	X =  248.562  mm,	Y =   -335.401  mm,	Z =   -309.100  mm,
	W =  90.000 deg,	P =   0.000 deg,	R =   90.000 deg
};
P[1872]{
   GP1:
	UF : 0, UT : 6,		CONFIG : 'N U T, 0, 0, 0',
	X =  247.422  mm,	Y =   -335.745  mm,	Z =   -309.000  mm,
	W =  90.000 deg,	P =   0.000 deg,	R =   90.000 deg
};
P[1873]{
   GP1:
	UF : 0, UT : 6,		CONFIG : 'N U T, 0, 0, 0',
	X =  247.235  mm,	Y =   -336.680  mm,	Z =   -320.106  mm,
	W =  90.000 deg,	P =   0.000 deg,	R =   90.000 deg
};
P[1874]{
   GP1:
	UF : 0, UT : 6,		CONFIG : 'N U T, 0, 0, 0',
	X =  245.967  mm,	Y =   -336.637  mm,	Z =   -309.000  mm,
	W =  90.000 deg,	P =   0.000 deg,	R =   90.000 deg
};
P[1875]{
   GP1:
	UF : 0, UT : 6,		CONFIG : 'N U T, 0, 0, 0',
	X =  245.051  mm,	Y =   -337.530  mm,	Z =   -309.000  mm,
	W =  90.000 deg,	P =   0.000 deg,	R =   90.000 deg
};
P[1876]{
   GP1:
	UF : 0, UT : 6,		CONFIG : 'N U T, 0, 0, 0',
	X =  243.808  mm,	Y =   -338.459  mm,	Z =   -309.000  mm,
	W =  90.000 deg,	P =   0.000 deg,	R =   90.000 deg
};
P[1877]{
   GP1:
	UF : 0, UT : 6,		CONFIG : 'N U T, 0, 0, 0',
	X =  242.999  mm,	Y =   -338.641  mm,	Z =   -309.100  mm,
	W =  90.000 deg,	P =   0.000 deg,	R =   90.000 deg
};
P[1878]{
   GP1:
	UF : 0, UT : 6,		CONFIG : 'N U T, 0, 0, 0',
	X =  242.520  mm,	Y =   -339.408  mm,	Z =   -309.100  mm,
	W =  90.000 deg,	P =   0.000 deg,	R =   90.000 deg
};
P[1879]{
   GP1:
	UF : 0, UT : 6,		CONFIG : 'N U T, 0, 0, 0',
	X =  240.721  mm,	Y =   -340.006  mm,	Z =   -309.100  mm,
	W =  90.000 deg,	P =   0.000 deg,	R =   90.000 deg
};
P[1880]{
   GP1:
	UF : 0, UT : 6,		CONFIG : 'N U T, 0, 0, 0',
	X =  239.710  mm,	Y =   -340.345  mm,	Z =   -309.000  mm,
	W =  90.000 deg,	P =   0.000 deg,	R =   90.000 deg
};
P[1881]{
   GP1:
	UF : 0, UT : 6,		CONFIG : 'N U T, 0, 0, 0',
	X =  238.388  mm,	Y =   -341.396  mm,	Z =   -309.000  mm,
	W =  90.000 deg,	P =   0.000 deg,	R =   90.000 deg
};
P[1882]{
   GP1:
	UF : 0, UT : 6,		CONFIG : 'N U T, 0, 0, 0',
	X =  236.976  mm,	Y =   -342.451  mm,	Z =   -309.000  mm,
	W =  90.000 deg,	P =   0.000 deg,	R =   90.000 deg
};
P[1883]{
   GP1:
	UF : 0, UT : 6,		CONFIG : 'N U T, 0, 0, 0',
	X =  236.149  mm,	Y =   -342.418  mm,	Z =   -309.100  mm,
	W =  90.000 deg,	P =   0.000 deg,	R =   90.000 deg
};
P[1884]{
   GP1:
	UF : 0, UT : 6,		CONFIG : 'N U T, 0, 0, 0',
	X =  235.257  mm,	Y =   -343.142  mm,	Z =   -328.083  mm,
	W =  90.000 deg,	P =   0.000 deg,	R =   90.000 deg
};
P[1885]{
   GP1:
	UF : 0, UT : 6,		CONFIG : 'N U T, 0, 0, 0',
	X =  233.924  mm,	Y =   -343.541  mm,	Z =   -309.100  mm,
	W =  90.000 deg,	P =   0.000 deg,	R =   90.000 deg
};
P[1886]{
   GP1:
	UF : 0, UT : 6,		CONFIG : 'N U T, 0, 0, 0',
	X =  232.946  mm,	Y =   -344.617  mm,	Z =   -309.000  mm,
	W =  90.000 deg,	P =   0.000 deg,	R =   90.000 deg
};
P[1887]{
   GP1:
	UF : 0, UT : 6,		CONFIG : 'N U T, 0, 0, 0',
	X =  231.730  mm,	Y =   -344.591  mm,	Z =   -309.000  mm,
	W =  90.000 deg,	P =   0.000 deg,	R =   90.000 deg
};
P[1888]{
   GP1:
	UF : 0, UT : 6,		CONFIG : 'N U T, 0, 0, 0',
	X =  231.106  mm,	Y =   -345.617  mm,	Z =   -309.100  mm,
	W =  90.000 deg,	P =   0.000 deg,	R =   90.000 deg
};
P[1889]{
   GP1:
	UF : 0, UT : 6,		CONFIG : 'N U T, 0, 0, 0',
	X =  229.581  mm,	Y =   -346.237  mm,	Z =   -309.000  mm,
	W =  90.000 deg,	P =   0.000 deg,	R =   90.000 deg
};
P[1890]{
   GP1:
	UF : 0, UT : 6,		CONFIG : 'N U T, 0, 0, 0',
	X =  228.460  mm,	Y =   -346.775  mm,	Z =   -309.000  mm,
	W =  90.000 deg,	P =   0.000 deg,	R =   90.000 deg
};
P[1891]{
   GP1:
	UF : 0, UT : 6,		CONFIG : 'N U T, 0, 0, 0',
	X =  227.482  mm,	Y =   -347.579  mm,	Z =   -309.000  mm,
	W =  90.000 deg,	P =   0.000 deg,	R =   90.000 deg
};
P[1892]{
   GP1:
	UF : 0, UT : 6,		CONFIG : 'N U T, 0, 0, 0',
	X =  226.728  mm,	Y =   -348.283  mm,	Z =   -309.000  mm,
	W =  90.000 deg,	P =   0.000 deg,	R =   90.000 deg
};
P[1893]{
   GP1:
	UF : 0, UT : 6,		CONFIG : 'N U T, 0, 0, 0',
	X =  225.408  mm,	Y =   -348.579  mm,	Z =   -309.000  mm,
	W =  90.000 deg,	P =   0.000 deg,	R =   90.000 deg
};
P[1894]{
   GP1:
	UF : 0, UT : 6,		CONFIG : 'N U T, 0, 0, 0',
	X =  224.991  mm,	Y =   -349.488  mm,	Z =   -309.100  mm,
	W =  90.000 deg,	P =   0.000 deg,	R =   90.000 deg
};
P[1895]{
   GP1:
	UF : 0, UT : 6,		CONFIG : 'N U T, 0, 0, 0',
	X =  223.968  mm,	Y =   -349.539  mm,	Z =   -309.000  mm,
	W =  90.000 deg,	P =   0.000 deg,	R =   90.000 deg
};
P[1896]{
   GP1:
	UF : 0, UT : 6,		CONFIG : 'N U T, 0, 0, 0',
	X =  223.129  mm,	Y =   -350.051  mm,	Z =   -314.213  mm,
	W =  90.000 deg,	P =   0.000 deg,	R =   90.000 deg
};
P[1897]{
   GP1:
	UF : 0, UT : 6,		CONFIG : 'N U T, 0, 0, 0',
	X =  222.469  mm,	Y =   -350.654  mm,	Z =   -309.577  mm,
	W =  90.000 deg,	P =   0.000 deg,	R =   90.000 deg
};
P[1898]{
   GP1:
	UF : 0, UT : 6,		CONFIG : 'N U T, 0, 0, 0',
	X =  221.386  mm,	Y =   -350.938  mm,	Z =   -309.100  mm,
	W =  90.000 deg,	P =   0.000 deg,	R =   90.000 deg
};
P[1899]{
   GP1:
	UF : 0, UT : 6,		CONFIG : 'N U T, 0, 0, 0',
	X =  220.623  mm,	Y =   -351.619  mm,	Z =   -309.000  mm,
	W =  90.000 deg,	P =   0.000 deg,	R =   90.000 deg
};
P[1900]{
   GP1:
	UF : 0, UT : 6,		CONFIG : 'N U T, 0, 0, 0',
	X =  219.642  mm,	Y =   -352.592  mm,	Z =   -321.382  mm,
	W =  90.000 deg,	P =   0.000 deg,	R =   90.000 deg
};
P[1901]{
   GP1:
	UF : 0, UT : 6,		CONFIG : 'N U T, 0, 0, 0',
	X =  218.872  mm,	Y =   -352.238  mm,	Z =   -309.000  mm,
	W =  90.000 deg,	P =   0.000 deg,	R =   90.000 deg
};
P[1902]{
   GP1:
	UF : 0, UT : 6,		CONFIG : 'N U T, 0, 0, 0',
	X =  218.325  mm,	Y =   -353.159  mm,	Z =   -309.000  mm,
	W =  90.000 deg,	P =   0.000 deg,	R =   90.000 deg
};
P[1903]{
   GP1:
	UF : 0, UT : 6,		CONFIG : 'N U T, 0, 0, 0',
	X =  217.117  mm,	Y =   -353.353  mm,	Z =   -309.000  mm,
	W =  90.000 deg,	P =   0.000 deg,	R =   90.000 deg
};
P[1904]{
   GP1:
	UF : 0, UT : 6,		CONFIG : 'N U T, 0, 0, 0',
	X =  216.830  mm,	Y =   -354.032  mm,	Z =   -309.000  mm,
	W =  90.000 deg,	P =   0.000 deg,	R =   90.000 deg
};
P[1905]{
   GP1:
	UF : 0, UT : 6,		CONFIG : 'N U T, 0, 0, 0',
	X =  215.180  mm,	Y =   -354.468  mm,	Z =   -317.962  mm,
	W =  90.000 deg,	P =   0.000 deg,	R =   90.000 deg
};
P[1906]{
   GP1:
	UF : 0, UT : 6,		CONFIG : 'N U T, 0, 0, 0',
	X =  213.998  mm,	Y =   -355.496  mm,	Z =   -309.000  mm,
	W =  90.000 deg,	P =   0.000 deg,	R =   90.000 deg
};
P[1907]{
   GP1:
	UF : 0, UT : 6,		CONFIG : 'N U T, 0, 0, 0',
	X =  212.895  mm,	Y =   -355.957  mm,	Z =   -309.000  mm,
	W =  90.000 deg,	P =   0.000 deg,	R =   90.000 deg
};
P[1908]{
   GP1:
	UF : 0, UT : 6,		CONFIG : 'N U T, 0, 0, 0',
	X =  212.166  mm,	Y =   -356.433  mm,	Z =   -309.100  mm,
	W =  90.000 deg,	P =   0.000 deg,	R =   90.000 deg
};
P[1909]{
   GP1:
	UF : 0, UT : 6,		CONFIG : 'N U T, 0, 0, 0',
	X =  211.060  mm,	Y =   -356.896  mm,	Z =   -309.100  mm,
	W =  90.000 deg,	P =   0.000 deg,	R =   90.000 deg
};
P[1910]{
   GP1:
	UF : 0, UT : 6,		CONFIG : 'N U T, 0, 0, 0',
	X =  209.472  mm,	Y =   -358.263  mm,	Z =   -309.000  mm,
	W =  90.000 deg,	P =   0.000 deg,	R =   90.000 deg
};
P[1911]{
   GP1:
	UF : 0, UT : 6,		CONFIG : 'N U T, 0, 0, 0',
	X =  208.197  mm,	Y =   -358.550  mm,	Z =   -309.000  mm,
	W =  90.000 deg,	P =   0.000 deg,	R =   90.000 deg
};
P[1912]{
   GP1:
	UF : 0, UT : 6,		CONFIG : 'N U T, 0, 0, 0',
	X =  207.007  mm,	Y =   -359.434  mm,	Z =   -309.000  mm,
	W =  90.000 deg,	P =   0.000 deg,	R =   90.000 deg
};
P[1913]{
   GP1:
	UF : 0, UT : 6,		CONFIG : 'N U T, 0, 0, 0',
	X =  206.131  mm,	Y =   -360.046  mm,	Z =   -309.000  mm,
	W =  90.000 deg,	P =   0.000 deg,	R =   90.000 deg
};
P[1914]{
   GP1:
	UF : 0, UT : 6,		CONFIG : 'N U T, 0, 0, 0',
	X =  205.000  mm,	Y =   -360.301  mm,	Z =   -309.100  mm,
	W =  90.000 deg,	P =   0.000 deg,	R =   90.000 deg
};
P[1915]{
   GP1:
	UF : 0, UT : 6,		CONFIG : 'N U T, 0, 0, 0',
	X =  204.421  mm,	Y =   -361.260  mm,	Z =   -309.000  mm,
	W =  90.000 deg,	P =   0.000 deg,	R =   90.000 deg
};
P[1916]{
   GP1:
	UF : 0, UT : 6,		CONFIG : 'N U T, 0, 0, 0',
	X =  202.482  mm,	Y =   -361.984  mm,	Z =   -309.100  mm,
	W =  90.000 deg,	P =   0.000 deg,	R =   90.000 deg
};
P[1917]{
   GP1:
	UF : 0, UT : 6,		CONFIG : 'N U T, 0, 0, 0',
	X =  201.337  mm,	Y =   -362.133  mm,	Z =   -309.115  mm,
	W =  90.000 deg,	P =   0.000 deg,	R =   90.000 deg
};
P[1918]{
   GP1:
	UF : 0, UT : 6,		CONFIG : 'N U T, 0, 0, 0',
	X =  200.951  mm,	Y =   -362.839  mm,	Z =   -309.100  mm,
	W =  90.000 deg,	P =   0.000 deg,	R =   90.000 deg
};
P[1919]{
   GP1:
	UF : 0, UT : 6,		CONFIG : 'N U T, 0, 0, 0',
	X =  199.770  mm,	Y =   -363.436  mm,	Z =   -309.100  mm,
	W =  90.000 deg,	P =   0.000 deg,	R =   90.000 deg
};
P[1920]{
   GP1:
	UF : 0, UT : 6,		CONFIG : 'N U T, 0, 0, 0',
	X =  198.938  mm,	Y =   -363.987  mm,	Z =   -309.100  mm,
	W =  90.000 deg,	P =   0.000 deg,	R =   90.000 deg
};
P[1921]{
   GP1:
	UF : 0, UT : 6,		CONFIG : 'N U T, 0, 0, 0',
	X =  198.274  mm,	Y =   -364.327  mm,	Z =   -309.000  mm,
	W =  90.000 deg,	P =   0.000 deg,	R =   90.000 deg
};
P[1922]{
   GP1:
	UF : 0, UT : 6,		CONFIG : 'N U T, 0, 0, 0',
	X =  197.346  mm,	Y =   -364.943  mm,	Z =   -313.498  mm,
	W =  90.000 deg,	P =   0.000 deg,	R =   90.000 deg
};
P[1923]{
   GP1:
	UF : 0, UT : 6,		CONFIG : 'N U T, 0, 0, 0',
	X =  196.755  mm,	Y =   -365.858  mm,	Z =   -309.000  mm,
	W =  90.000 deg,	P =   0.000 deg,	R =   90.000 deg
};
P[1924]{
   GP1:
	UF : 0, UT : 6,		CONFIG : 'N U T, 0, 0, 0',
	X =  196.093  mm,	Y =   -366.179  mm,	Z =   -309.000  mm,
	W =  90.000 deg,	P =   0.000 deg,	R =   90.000 deg
};
P[1925]{
   GP1:
	UF : 0, UT : 6,		CONFIG : 'N U T, 0, 0, 0',
	X =  194.785  mm,	Y =   -366.104  mm,	Z =   -309.100  mm,
	W =  90.000 deg,	P =   0.000 deg,	R =   90.000 deg
};
P[1926]{
   GP1:
	UF : 0, UT : 6,		CONFIG : 'N U T, 0, 0, 0',
	X =  193.345  mm,	Y =   -367.474  mm,	Z =   -309.000  mm,
	W =  90.000 deg,	P =   0.000 deg,	R =   90.000 deg
};
P[1927]{
   GP1:
	UF : 0, UT : 6,		CONFIG : 'N U T, 0, 0, 0',
	X =  192.179  mm,	Y =   -367.513  mm,	Z =   -316.834  mm,
	W =  90.000 deg,	P =   0.000 deg,	R =   90.000 deg
};
P[1928]{
   GP1:
	UF : 0, UT : 6,		CONFIG : 'N U T, 0, 0, 0',
	X =  191.363  mm,	Y =   -368.920  mm,	Z =   -318.857  mm,
	W =  90.000 deg,	P =   0.000 deg,	R =   90.000 deg
};
P[1929]{
   GP1:
	UF : 0, UT : 6,		CONFIG : 'N U T, 0, 0, 0',
	X =  190.046  mm,	Y =   -369.124  mm,	Z =   -309.000  mm,
	W =  90.000 deg,	P =   0.000 deg,	R =   90.000 deg
};
P[1930]{
   GP1:
	UF : 0, UT : 6,		CONFIG : 'N U T, 0, 0, 0',
	X =  188.428  mm,	Y =   -369.682  mm,	Z =   -309.000  mm,
	W =  90.000 deg,	P =   0.000 deg,	R =   90.000 deg
};
P[1931]{
   GP1:
	UF : 0, UT : 6,		CONFIG : 'N U T, 0, 0, 0',
	X =  187.625  mm,	Y =   -370.456  mm,	Z =   -309.000  mm,
	W =  90.000 deg,	P =   0.000 deg,	R =   90.000 deg
};
P[1932]{
   GP1:
	UF : 0, UT : 6,		CONFIG : 'N U T, 0, 0, 0',
	X =  186.427  mm,	Y =   -371.699  mm,	Z =   -312.203  mm,
	W =  90.000 deg,	P =   0.000 deg,	R =   90.000 deg
};
P[1933]{
   GP1:
	UF : 0, UT : 6,		CONFIG : 'N U T, 0, 0, 0',
	X =  185.466  mm,	Y =   -371.863  mm,	Z =   -309.100  mm,
	W =  90.000 deg,	P =   0.000 deg,	R =   90.000 deg
};
P[1934]{
   GP1:
	UF : 0, UT : 6,		CONFIG : 'N U T, 0, 0, 0',
	X =  184.245  mm,	Y =   -372.318  mm,	Z =   -309.000  mm,
	W =  90.000 deg,	P =   0.000 deg,	R =   90.000 deg
};
P[1935]{
   GP1:
	UF : 0, UT : 6,		CONFIG : 'N U T, 0, 0, 0',
	X =  183.685  mm,	Y =   -372.780  mm,	Z =   -309.100  mm,
	W =  90.000 deg,	P =   0.000 deg,	R =   90.000 deg
};
P[1936]{
   GP1:
	UF : 0, UT : 6,		CONFIG : 'N U T, 0, 0, 0',
	X =  183.047  mm,	Y =   -373.648  mm,	Z =   -309.000  mm,
	W =  90.000 deg,	P =   0.000 deg,	R =   90.000 deg
};
P[1937]{
   GP1:
	UF : 0, UT : 6,		CONFIG : 'N U T, 0, 0, 0',
	X =  182.264  mm,	Y =   -374.207  mm,	Z =   -309.000  mm,
	W =  90.000 deg,	P =   0.000 deg,	R =   90.000 deg
};
P[1938]{
   GP1:
	UF : 0, UT : 6,		CONFIG : 'N U T, 0, 0, 0',
	X =  180.861  mm,	Y =   -374.555  mm,	Z =   -309.000  mm,
	W =  90.000 deg,	P =   0.000 deg,	R =   90.000 deg
};
P[1939]{
   GP1:
	UF : 0, UT : 6,		CONFIG : 'N U T, 0, 0, 0',
	X =  180.053  mm,	Y =   -374.605  mm,	Z =   -309.000  mm,
	W =  90.000 deg,	P =   0.000 deg,	R =   90.000 deg
};
P[1940]{
   GP1:
	UF : 0, UT : 6,		CONFIG : 'N U T, 0, 0, 0',
	X =  178.977  mm,	Y =   -375.401  mm,	Z =   -309.000  mm,
	W =  90.000 deg,	P =   0.000 deg,	R =   90.000 deg
};
P[1941]{
   GP1:
	UF : 0, UT : 6,		CONFIG : 'N U T, 0, 0, 0',
	X =  178.071  mm,	Y =   -375.997  mm,	Z =   -309.100  mm,
	W =  90.000 deg,	P =   0.000 deg,	R =   90.000 deg
};
P[1942]{
   GP1:
	UF : 0, UT : 6,		CONFIG : 'N U T, 0, 0, 0',
	X =  176.472  mm,	Y =   -376.780  mm,	Z =   -319.410  mm,
	W =  90.000 deg,	P =   0.000 deg,	R =   90.000 deg
};
P[1943]{
   GP1:
	UF : 0, UT : 6,		CONFIG : 'N U T, 0, 0, 0',
	X =  175.518  mm,	Y =   -377.434  mm,	Z =   -318.225  mm,
	W =  90.000 deg,	P =   0.000 deg,	R =   90.000 deg
};
P[1944]{
   GP1:
	UF : 0, UT : 6,		CONFIG : 'N U T, 0, 0, 0',
	X =  174.768  mm,	Y =   -377.867  mm,	Z =   -309.100  mm,
	W =  90.000 deg,	P =   0.000 deg,	R =   90.000 deg
};
P[1945]{
   GP1:
	UF : 0, UT : 6,		CONFIG : 'N U T, 0, 0, 0',
	X =  174.000  mm,	Y =   -377.913  mm,	Z =   -309.000  mm,
	W =  90.000 deg,	P =   0.000 deg,	R =   90.000 deg
};
P[1946]{
   GP1:
	UF : 0, UT : 6,		CONFIG : 'N U T, 0, 0, 0',
	X =  173.393  mm,	Y =   -378.705  mm,	Z =   -309.100  mm,
	W =  90.000 deg,	P =   0.000 deg,	R =   90.000 deg
};
P[1947]{
   GP1:
	UF : 0, UT : 6,		CONFIG : 'N U T, 0, 0, 0',
	X =  172.740  mm,	Y =   -379.505  mm,	Z =   -309.000  mm,
	W =  90.000 deg,	P =   0.000 deg,	R =   90.000 deg
};
P[1948]{
   GP1:
	UF : 0, UT : 6,		CONFIG : 'N U T, 0, 0, 0',
	X =  171.553  mm,	Y =   -379.511  mm,	Z =   -309.000  mm,
	W =  90.000 deg,	P =   0.000 deg,	R =   90.000 deg
};
P[1949]{
   GP1:
	UF : 0, UT : 6,		CONFIG : 'N U T, 0, 0, 0',
	X =  170.266  mm,	Y =   -380.690  mm,	Z =   -309.100  mm,
	W =  90.000 deg,	P =   0.000 deg,	R =   90.000 deg
};
P[1950]{
   GP1:
	UF : 0, UT : 6,		CONFIG : 'N U T, 0, 0, 0',
	X =  169.463  mm,	Y =   -381.050  mm,	Z =   -309.100  mm,
	W =  90.000 deg,	P =   0.000 deg,	R =   90.000 deg
};
P[1951]{
   GP1:
	UF : 0, UT : 6,		CONFIG : 'N U T, 0, 0, 0',
	X =  168.875  mm,	Y =   -381.396  mm,	Z =   -309.000  mm,
	W =  90.000 deg,	P =   0.000 deg,	R =   90.000 deg
};
P[1952]{
   GP1:
	UF : 0, UT : 6,		CONFIG : 'N U T, 0, 0, 0',
	X =  168.134  mm,	Y =   -381.604  mm,	Z =   -309.100  mm,
	W =  90.000 deg,	P =   0.000 deg,	R =   90.000 deg
};
P[1953]{
   GP1:
	UF : 0, UT : 6,		CONFIG : 'N U T, 0, 0, 0',
	X =  167.049  mm,	Y =   -382.254  mm,	Z =   -309.000  mm,
	W =  90.000 deg,	P =   0.000 deg,	R =   90.000 deg
};
P[1954]{
   GP1:
	UF : 0, UT : 6,		CONFIG : 'N U T, 0, 0, 0',
	X =  166.356  mm,	Y =   -382.864  mm,	Z =   -319.959  mm,
	W =  90.000 deg,	P =   0.000 deg,	R =   90.000 deg
};
P[1955]{
   GP1:
	UF : 0, UT : 6,		CONFIG : 'N U T, 0, 0, 0',
	X =  165.358  mm,	Y =   -383.111  mm,	Z =   -309.100  mm,
	W =  90.000 deg,	P =   0.000 deg,	R =   90.000 deg
};
P[1956]{
   GP1:
	UF : 0, UT : 6,		CONFIG : 'N U T, 0, 0, 0',
	X =  164.331  mm,	Y =   -384.035  mm,	Z =   -309.000  mm,
	W =  90.000 deg,	P =   0.000 deg,	R =   90.000 deg
};
P[1957]{
   GP1:
	UF : 0, UT : 6,		CONFIG : 'N U T, 0, 0, 0',
	X =  163.613  mm,	Y =   -384.424  mm,	Z =   -309.100  mm,
	W =  90.000 deg,	P =   0.000 deg,	R =   90.000 deg
};
P[1958]{
   GP1:
	UF : 0, UT : 6,		CONFIG : 'N U T, 0, 0, 0',
	X =  162.736  mm,	Y =   -384.918  mm,	Z =   -309.100  mm,
	W =  90.000 deg,	P =   0.000 deg,	R =   90.000 deg
};
P[1959]{
   GP1:
	UF : 0, UT : 6,		CONFIG : 'N U T, 0, 0, 0',
	X =  162.209  mm,	Y =   -385.446  mm,	Z =   -309.050  mm,
	W =  90.000 deg,	P =   0.000 deg,	R =   90.000 deg
};
P[1960]{
   GP1:
	UF : 0, UT : 6,		CONFIG : 'N U T, 0, 0, 0',
	X =  160.970  mm,	Y =   -386.136  mm,	Z =   -309.000  mm,
	W =  90.000 deg,	P =   0.000 deg,	R =   90.000 deg
};
P[1961]{
   GP1:
	UF : 0, UT : 6,		CONFIG : 'N U T, 0, 0, 0',
	X =  159.328  mm,	Y =   -386.935  mm,	Z =   -317.393  mm,
	W =  90.000 deg,	P =   0.000 deg,	R =   90.000 deg
};
P[1962]{
   GP1:
	UF : 0, UT : 6,		CONFIG : 'N U T, 0, 0, 0',
	X =  158.454  mm,	Y =   -387.478  mm,	Z =   -309.000  mm,
	W =  90.000 deg,	P =   0.000 deg,	R =   90.000 deg
};
P[1963]{
   GP1:
	UF : 0, UT : 6,		CONFIG : 'N U T, 0, 0, 0',
	X =  157.813  mm,	Y =   -388.057  mm,	Z =   -309.000  mm,
	W =  90.000 deg,	P =   0.000 deg,	R =   90.000 deg
};
P[1964]{
   GP1:
	UF : 0, UT : 6,		CONFIG : 'N U T, 0, 0, 0',
	X =  156.616  mm,	Y =   -388.189  mm,	Z =   -309.100  mm,
	W =  90.000 deg,	P =   0.000 deg,	R =   90.000 deg
};
P[1965]{
   GP1:
	UF : 0, UT : 6,		CONFIG : 'N U T, 0, 0, 0',
	X =  155.251  mm,	Y =   -388.814  mm,	Z =   -309.100  mm,
	W =  90.000 deg,	P =   0.000 deg,	R =   90.000 deg
};
P[1966]{
   GP1:
	UF : 0, UT : 6,		CONFIG : 'N U T, 0, 0, 0',
	X =  154.672  mm,	Y =   -389.734  mm,	Z =   -309.000  mm,
	W =  90.000 deg,	P =   0.000 deg,	R =   90.000 deg
};
P[1967]{
   GP1:
	UF : 0, UT : 6,		CONFIG : 'N U T, 0, 0, 0',
	X =  153.912  mm,	Y =   -389.865  mm,	Z =   -309.000  mm,
	W =  90.000 deg,	P =   0.000 deg,	R =   90.000 deg
};
P[1968]{
   GP1:
	UF : 0, UT : 6,		CONFIG : 'N U T, 0, 0, 0',
	X =  153.303  mm,	Y =   -390.841  mm,	Z =   -309.000  mm,
	W =  90.000 deg,	P =   0.000 deg,	R =   90.000 deg
};
P[1969]{
   GP1:
	UF : 0, UT : 6,		CONFIG : 'N U T, 0, 0, 0',
	X =  151.916  mm,	Y =   -391.243  mm,	Z =   -309.000  mm,
	W =  90.000 deg,	P =   0.000 deg,	R =   90.000 deg
};
P[1970]{
   GP1:
	UF : 0, UT : 6,		CONFIG : 'N U T, 0, 0, 0',
	X =  151.066  mm,	Y =   -392.066  mm,	Z =   -309.000  mm,
	W =  90.000 deg,	P =   0.000 deg,	R =   90.000 deg
};
P[1971]{
   GP1:
	UF : 0, UT : 6,		CONFIG : 'N U T, 0, 0, 0',
	X =  149.784  mm,	Y =   -392.830  mm,	Z =   -309.100  mm,
	W =  90.000 deg,	P =   0.000 deg,	R =   90.000 deg
};
P[1972]{
   GP1:
	UF : 0, UT : 6,		CONFIG : 'N U T, 0, 0, 0',
	X =  148.664  mm,	Y =   -392.829  mm,	Z =   -309.100  mm,
	W =  90.000 deg,	P =   0.000 deg,	R =   90.000 deg
};
P[1973]{
   GP1:
	UF : 0, UT : 6,		CONFIG : 'N U T, 0, 0, 0',
	X =  147.712  mm,	Y =   -393.864  mm,	Z =   -309.000  mm,
	W =  90.000 deg,	P =   0.000 deg,	R =   90.000 deg
};
P[1974]{
   GP1:
	UF : 0, UT : 6,		CONFIG : 'N U T, 0, 0, 0',
	X =  146.950  mm,	Y =   -393.960  mm,	Z =   -309.000  mm,
	W =  90.000 deg,	P =   0.000 deg,	R =   90.000 deg
};
P[1975]{
   GP1:
	UF : 0, UT : 6,		CONFIG : 'N U T, 0, 0, 0',
	X =  146.208  mm,	Y =   -394.773  mm,	Z =   -309.000  mm,
	W =  90.000 deg,	P =   0.000 deg,	R =   90.000 deg
};
P[1976]{
   GP1:
	UF : 0, UT : 6,		CONFIG : 'N U T, 0, 0, 0',
	X =  145.184  mm,	Y =   -394.852  mm,	Z =   -309.100  mm,
	W =  90.000 deg,	P =   0.000 deg,	R =   90.000 deg
};
P[1977]{
   GP1:
	UF : 0, UT : 6,		CONFIG : 'N U T, 0, 0, 0',
	X =  143.553  mm,	Y =   -395.880  mm,	Z =   -309.000  mm,
	W =  90.000 deg,	P =   0.000 deg,	R =   90.000 deg
};
P[1978]{
   GP1:
	UF : 0, UT : 6,		CONFIG : 'N U T, 0, 0, 0',
	X =  142.760  mm,	Y =   -396.576  mm,	Z =   -309.100  mm,
	W =  90.000 deg,	P =   0.000 deg,	R =   90.000 deg
};
P[1979]{
   GP1:
	UF : 0, UT : 6,		CONFIG : 'N U T, 0, 0, 0',
	X =  140.503  mm,	Y =   -397.919  mm,	Z =   -309.100  mm,
	W =  90.000 deg,	P =   0.000 deg,	R =   90.000 deg
};
P[1980]{
   GP1:
	UF : 0, UT : 6,		CONFIG : 'N U T, 0, 0, 0',
	X =  139.521  mm,	Y =   -398.012  mm,	Z =   -309.100  mm,
	W =  90.000 deg,	P =   0.000 deg,	R =   90.000 deg
};
P[1981]{
   GP1:
	UF : 0, UT : 6,		CONFIG : 'N U T, 0, 0, 0',
	X =  138.640  mm,	Y =   -398.575  mm,	Z =   -309.000  mm,
	W =  90.000 deg,	P =   0.000 deg,	R =   90.000 deg
};
P[1982]{
   GP1:
	UF : 0, UT : 6,		CONFIG : 'N U T, 0, 0, 0',
	X =  137.549  mm,	Y =   -399.589  mm,	Z =   -309.000  mm,
	W =  90.000 deg,	P =   0.000 deg,	R =   90.000 deg
};
P[1983]{
   GP1:
	UF : 0, UT : 6,		CONFIG : 'N U T, 0, 0, 0',
	X =  136.858  mm,	Y =   -400.280  mm,	Z =   -309.000  mm,
	W =  90.000 deg,	P =   0.000 deg,	R =   90.000 deg
};
P[1984]{
   GP1:
	UF : 0, UT : 6,		CONFIG : 'N U T, 0, 0, 0',
	X =  135.718  mm,	Y =   -400.452  mm,	Z =   -309.000  mm,
	W =  90.000 deg,	P =   0.000 deg,	R =   90.000 deg
};
P[1985]{
   GP1:
	UF : 0, UT : 6,		CONFIG : 'N U T, 0, 0, 0',
	X =  134.677  mm,	Y =   -401.299  mm,	Z =   -309.000  mm,
	W =  90.000 deg,	P =   0.000 deg,	R =   90.000 deg
};
P[1986]{
   GP1:
	UF : 0, UT : 6,		CONFIG : 'N U T, 0, 0, 0',
	X =  133.827  mm,	Y =   -401.414  mm,	Z =   -309.000  mm,
	W =  90.000 deg,	P =   0.000 deg,	R =   90.000 deg
};
P[1987]{
   GP1:
	UF : 0, UT : 6,		CONFIG : 'N U T, 0, 0, 0',
	X =  133.368  mm,	Y =   -402.189  mm,	Z =   -309.000  mm,
	W =  90.000 deg,	P =   0.000 deg,	R =   90.000 deg
};
P[1988]{
   GP1:
	UF : 0, UT : 6,		CONFIG : 'N U T, 0, 0, 0',
	X =  132.709  mm,	Y =   -402.717  mm,	Z =   -309.000  mm,
	W =  90.000 deg,	P =   0.000 deg,	R =   90.000 deg
};
P[1989]{
   GP1:
	UF : 0, UT : 6,		CONFIG : 'N U T, 0, 0, 0',
	X =  131.281  mm,	Y =   -403.108  mm,	Z =   -309.000  mm,
	W =  90.000 deg,	P =   0.000 deg,	R =   90.000 deg
};
P[1990]{
   GP1:
	UF : 0, UT : 6,		CONFIG : 'N U T, 0, 0, 0',
	X =  130.231  mm,	Y =   -403.479  mm,	Z =   -309.100  mm,
	W =  90.000 deg,	P =   0.000 deg,	R =   90.000 deg
};
P[1991]{
   GP1:
	UF : 0, UT : 6,		CONFIG : 'N U T, 0, 0, 0',
	X =  129.597  mm,	Y =   -404.057  mm,	Z =   -309.000  mm,
	W =  90.000 deg,	P =   0.000 deg,	R =   90.000 deg
};
P[1992]{
   GP1:
	UF : 0, UT : 6,		CONFIG : 'N U T, 0, 0, 0',
	X =  128.443  mm,	Y =   -404.240  mm,	Z =   -309.100  mm,
	W =  90.000 deg,	P =   0.000 deg,	R =   90.000 deg
};
P[1993]{
   GP1:
	UF : 0, UT : 6,		CONFIG : 'N U T, 0, 0, 0',
	X =  127.871  mm,	Y =   -405.193  mm,	Z =   -309.100  mm,
	W =  90.000 deg,	P =   0.000 deg,	R =   90.000 deg
};
P[1994]{
   GP1:
	UF : 0, UT : 6,		CONFIG : 'N U T, 0, 0, 0',
	X =  126.940  mm,	Y =   -405.360  mm,	Z =   -309.000  mm,
	W =  90.000 deg,	P =   0.000 deg,	R =   90.000 deg
};
P[1995]{
   GP1:
	UF : 0, UT : 6,		CONFIG : 'N U T, 0, 0, 0',
	X =  126.733  mm,	Y =   -406.117  mm,	Z =   -309.000  mm,
	W =  90.000 deg,	P =   0.000 deg,	R =   90.000 deg
};
P[1996]{
   GP1:
	UF : 0, UT : 6,		CONFIG : 'N U T, 0, 0, 0',
	X =  125.297  mm,	Y =   -406.512  mm,	Z =   -309.000  mm,
	W =  90.000 deg,	P =   0.000 deg,	R =   90.000 deg
};
P[1997]{
   GP1:
	UF : 0, UT : 6,		CONFIG : 'N U T, 0, 0, 0',
	X =  124.768  mm,	Y =   -407.328  mm,	Z =   -309.000  mm,
	W =  90.000 deg,	P =   0.000 deg,	R =   90.000 deg
};
P[1998]{
   GP1:
	UF : 0, UT : 6,		CONFIG : 'N U T, 0, 0, 0',
	X =  124.005  mm,	Y =   -407.406  mm,	Z =   -320.838  mm,
	W =  90.000 deg,	P =   0.000 deg,	R =   90.000 deg
};
P[1999]{
   GP1:
	UF : 0, UT : 6,		CONFIG : 'N U T, 0, 0, 0',
	X =  122.791  mm,	Y =   -407.939  mm,	Z =   -309.000  mm,
	W =  90.000 deg,	P =   0.000 deg,	R =   90.000 deg
};
P[2000]{
   GP1:
	UF : 0, UT : 6,		CONFIG : 'N U T, 0, 0, 0',
	X =  121.376  mm,	Y =   -408.435  mm,	Z =   -309.000  mm,
	W =  90.000 deg,	P =   0.000 deg,	R =   90.000 deg
};
P[2001]{
   GP1:
	UF : 0, UT : 6,		CONFIG : 'N U T, 0, 0, 0',
	X =  120.680  mm,	Y =   -409.255  mm,	Z =   -309.000  mm,
	W =  90.000 deg,	P =   0.000 deg,	R =   90.000 deg
};
P[2002]{
   GP1:
	UF : 0, UT : 6,		CONFIG : 'N U T, 0, 0, 0',
	X =  120.231  mm,	Y =   -409.951  mm,	Z =   -309.000  mm,
	W =  90.000 deg,	P =   0.000 deg,	R =   90.000 deg
};
P[2003]{
   GP1:
	UF : 0, UT : 6,		CONFIG : 'N U T, 0, 0, 0',
	X =  119.307  mm,	Y =   -409.899  mm,	Z =   -309.000  mm,
	W =  90.000 deg,	P =   0.000 deg,	R =   90.000 deg
};
P[2004]{
   GP1:
	UF : 0, UT : 6,		CONFIG : 'N U T, 0, 0, 0',
	X =  118.398  mm,	Y =   -410.962  mm,	Z =   -309.000  mm,
	W =  90.000 deg,	P =   0.000 deg,	R =   90.000 deg
};
P[2005]{
   GP1:
	UF : 0, UT : 6,		CONFIG : 'N U T, 0, 0, 0',
	X =  117.703  mm,	Y =   -410.902  mm,	Z =   -316.789  mm,
	W =  90.000 deg,	P =   0.000 deg,	R =   90.000 deg
};
P[2006]{
   GP1:
	UF : 0, UT : 6,		CONFIG : 'N U T, 0, 0, 0',
	X =  116.784  mm,	Y =   -411.144  mm,	Z =   -309.100  mm,
	W =  90.000 deg,	P =   0.000 deg,	R =   90.000 deg
};
P[2007]{
   GP1:
	UF : 0, UT : 6,		CONFIG : 'N U T, 0, 0, 0',
	X =  189.890  mm,	Y =   -369.869  mm,	Z =   -309.100  mm,
	W =  90.000 deg,	P =   0.000 deg,	R =   90.000 deg
};
P[2008]{
   GP1:
	UF : 0, UT : 6,		CONFIG : 'N U T, 0, 0, 0',
	X =  296.292  mm,	Y =   -325.746  mm,	Z =   -309.100  mm,
	W =  90.000 deg,	P =   0.000 deg,	R =   90.000 deg
};
P[2009]{
   GP1:
	UF : 0, UT : 6,		CONFIG : 'N U T, 0, 0, 0',
	X =  294.854  mm,	Y =   -326.018  mm,	Z =   -309.000  mm,
	W =  90.000 deg,	P =   0.000 deg,	R =   90.000 deg
};
P[2010]{
   GP1:
	UF : 0, UT : 6,		CONFIG : 'N U T, 0, 0, 0',
	X =  293.287  mm,	Y =   -327.087  mm,	Z =   -309.000  mm,
	W =  90.000 deg,	P =   0.000 deg,	R =   90.000 deg
};
P[2011]{
   GP1:
	UF : 0, UT : 6,		CONFIG : 'N U T, 0, 0, 0',
	X =  292.218  mm,	Y =   -327.512  mm,	Z =   -309.100  mm,
	W =  90.000 deg,	P =   0.000 deg,	R =   90.000 deg
};
P[2012]{
   GP1:
	UF : 0, UT : 6,		CONFIG : 'N U T, 0, 0, 0',
	X =  290.604  mm,	Y =   -328.546  mm,	Z =   -309.000  mm,
	W =  90.000 deg,	P =   0.000 deg,	R =   90.000 deg
};
P[2013]{
   GP1:
	UF : 0, UT : 6,		CONFIG : 'N U T, 0, 0, 0',
	X =  288.867  mm,	Y =   -329.278  mm,	Z =   -309.000  mm,
	W =  90.000 deg,	P =   0.000 deg,	R =   90.000 deg
};
P[2014]{
   GP1:
	UF : 0, UT : 6,		CONFIG : 'N U T, 0, 0, 0',
	X =  287.861  mm,	Y =   -329.931  mm,	Z =   -309.000  mm,
	W =  90.000 deg,	P =   0.000 deg,	R =   90.000 deg
};
P[2015]{
   GP1:
	UF : 0, UT : 6,		CONFIG : 'N U T, 0, 0, 0',
	X =  286.838  mm,	Y =   -330.612  mm,	Z =   -309.000  mm,
	W =  90.000 deg,	P =   0.000 deg,	R =   90.000 deg
};
P[2016]{
   GP1:
	UF : 0, UT : 6,		CONFIG : 'N U T, 0, 0, 0',
	X =  286.166  mm,	Y =   -331.329  mm,	Z =   -309.000  mm,
	W =  90.000 deg,	P =   0.000 deg,	R =   90.000 deg
};
P[2017]{
   GP1:
	UF : 0, UT : 6,		CONFIG : 'N U T, 0, 0, 0',
	X =  285.276  mm,	Y =   -331.778  mm,	Z =   -309.100  mm,
	W =  90.000 deg,	P =   0.000 deg,	R =   90.000 deg
};
P[2018]{
   GP1:
	UF : 0, UT : 6,		CONFIG : 'N U T, 0, 0, 0',
	X =  283.749  mm,	Y =   -332.698  mm,	Z =   -309.000  mm,
	W =  90.000 deg,	P =   0.000 deg,	R =   90.000 deg
};
P[2019]{
   GP1:
	UF : 0, UT : 6,		CONFIG : 'N U T, 0, 0, 0',
	X =  282.645  mm,	Y =   -333.429  mm,	Z =   -309.100  mm,
	W =  90.000 deg,	P =   0.000 deg,	R =   90.000 deg
};
P[2020]{
   GP1:
	UF : 0, UT : 6,		CONFIG : 'N U T, 0, 0, 0',
	X =  281.790  mm,	Y =   -333.720  mm,	Z =   -309.000  mm,
	W =  90.000 deg,	P =   0.000 deg,	R =   90.000 deg
};
P[2021]{
   GP1:
	UF : 0, UT : 6,		CONFIG : 'N U T, 0, 0, 0',
	X =  281.058  mm,	Y =   -333.870  mm,	Z =   -309.100  mm,
	W =  90.000 deg,	P =   0.000 deg,	R =   90.000 deg
};
P[2022]{
   GP1:
	UF : 0, UT : 6,		CONFIG : 'N U T, 0, 0, 0',
	X =  280.069  mm,	Y =   -334.629  mm,	Z =   -309.100  mm,
	W =  90.000 deg,	P =   0.000 deg,	R =   90.000 deg
};
P[2023]{
   GP1:
	UF : 0, UT : 6,		CONFIG : 'N U T, 0, 0, 0',
	X =  279.154  mm,	Y =   -334.563  mm,	Z =   -309.000  mm,
	W =  90.000 deg,	P =   0.000 deg,	R =   90.000 deg
};
P[2024]{
   GP1:
	UF : 0, UT : 6,		CONFIG : 'N U T, 0, 0, 0',
	X =  278.361  mm,	Y =   -334.972  mm,	Z =   -309.000  mm,
	W =  90.000 deg,	P =   0.000 deg,	R =   90.000 deg
};
P[2025]{
   GP1:
	UF : 0, UT : 6,		CONFIG : 'N U T, 0, 0, 0',
	X =  277.968  mm,	Y =   -336.200  mm,	Z =   -315.010  mm,
	W =  90.000 deg,	P =   0.000 deg,	R =   90.000 deg
};
P[2026]{
   GP1:
	UF : 0, UT : 6,		CONFIG : 'N U T, 0, 0, 0',
	X =  276.884  mm,	Y =   -336.602  mm,	Z =   -309.000  mm,
	W =  90.000 deg,	P =   0.000 deg,	R =   90.000 deg
};
P[2027]{
   GP1:
	UF : 0, UT : 6,		CONFIG : 'N U T, 0, 0, 0',
	X =  275.638  mm,	Y =   -336.912  mm,	Z =   -309.100  mm,
	W =  90.000 deg,	P =   0.000 deg,	R =   90.000 deg
};
P[2028]{
   GP1:
	UF : 0, UT : 6,		CONFIG : 'N U T, 0, 0, 0',
	X =  275.082  mm,	Y =   -337.523  mm,	Z =   -309.000  mm,
	W =  90.000 deg,	P =   0.000 deg,	R =   90.000 deg
};
P[2029]{
   GP1:
	UF : 0, UT : 6,		CONFIG : 'N U T, 0, 0, 0',
	X =  274.178  mm,	Y =   -337.531  mm,	Z =   -309.000  mm,
	W =  90.000 deg,	P =   0.000 deg,	R =   90.000 deg
};
P[2030]{
   GP1:
	UF : 0, UT : 6,		CONFIG : 'N U T, 0, 0, 0',
	X =  273.307  mm,	Y =   -338.512  mm,	Z =   -309.100  mm,
	W =  90.000 deg,	P =   0.000 deg,	R =   90.000 deg
};
P[2031]{
   GP1:
	UF : 0, UT : 6,		CONFIG : 'N U T, 0, 0, 0',
	X =  271.837  mm,	Y =   -338.826  mm,	Z =   -309.000  mm,
	W =  90.000 deg,	P =   0.000 deg,	R =   90.000 deg
};
P[2032]{
   GP1:
	UF : 0, UT : 6,		CONFIG : 'N U T, 0, 0, 0',
	X =  271.624  mm,	Y =   -339.739  mm,	Z =   -309.100  mm,
	W =  90.000 deg,	P =   0.000 deg,	R =   90.000 deg
};
P[2033]{
   GP1:
	UF : 0, UT : 6,		CONFIG : 'N U T, 0, 0, 0',
	X =  270.328  mm,	Y =   -340.219  mm,	Z =   -309.000  mm,
	W =  90.000 deg,	P =   0.000 deg,	R =   90.000 deg
};
P[2034]{
   GP1:
	UF : 0, UT : 6,		CONFIG : 'N U T, 0, 0, 0',
	X =  269.519  mm,	Y =   -340.506  mm,	Z =   -309.000  mm,
	W =  90.000 deg,	P =   0.000 deg,	R =   90.000 deg
};
P[2035]{
   GP1:
	UF : 0, UT : 6,		CONFIG : 'N U T, 0, 0, 0',
	X =  268.600  mm,	Y =   -341.036  mm,	Z =   -309.000  mm,
	W =  90.000 deg,	P =   0.000 deg,	R =   90.000 deg
};
P[2036]{
   GP1:
	UF : 0, UT : 6,		CONFIG : 'N U T, 0, 0, 0',
	X =  267.719  mm,	Y =   -341.573  mm,	Z =   -309.000  mm,
	W =  90.000 deg,	P =   0.000 deg,	R =   90.000 deg
};
P[2037]{
   GP1:
	UF : 0, UT : 6,		CONFIG : 'N U T, 0, 0, 0',
	X =  267.174  mm,	Y =   -342.268  mm,	Z =   -309.100  mm,
	W =  90.000 deg,	P =   0.000 deg,	R =   90.000 deg
};
P[2038]{
   GP1:
	UF : 0, UT : 6,		CONFIG : 'N U T, 0, 0, 0',
	X =  266.298  mm,	Y =   -342.675  mm,	Z =   -309.000  mm,
	W =  90.000 deg,	P =   0.000 deg,	R =   90.000 deg
};
P[2039]{
   GP1:
	UF : 0, UT : 6,		CONFIG : 'N U T, 0, 0, 0',
	X =  264.936  mm,	Y =   -343.351  mm,	Z =   -309.000  mm,
	W =  90.000 deg,	P =   0.000 deg,	R =   90.000 deg
};
P[2040]{
   GP1:
	UF : 0, UT : 6,		CONFIG : 'N U T, 0, 0, 0',
	X =  263.855  mm,	Y =   -344.025  mm,	Z =   -309.000  mm,
	W =  90.000 deg,	P =   0.000 deg,	R =   90.000 deg
};
P[2041]{
   GP1:
	UF : 0, UT : 6,		CONFIG : 'N U T, 0, 0, 0',
	X =  262.628  mm,	Y =   -344.584  mm,	Z =   -320.348  mm,
	W =  90.000 deg,	P =   0.000 deg,	R =   90.000 deg
};
P[2042]{
   GP1:
	UF : 0, UT : 6,		CONFIG : 'N U T, 0, 0, 0',
	X =  261.904  mm,	Y =   -345.057  mm,	Z =   -309.000  mm,
	W =  90.000 deg,	P =   0.000 deg,	R =   90.000 deg
};
P[2043]{
   GP1:
	UF : 0, UT : 6,		CONFIG : 'N U T, 0, 0, 0',
	X =  261.073  mm,	Y =   -345.842  mm,	Z =   -309.100  mm,
	W =  90.000 deg,	P =   0.000 deg,	R =   90.000 deg
};
P[2044]{
   GP1:
	UF : 0, UT : 6,		CONFIG : 'N U T, 0, 0, 0',
	X =  260.229  mm,	Y =   -346.116  mm,	Z =   -309.100  mm,
	W =  90.000 deg,	P =   0.000 deg,	R =   90.000 deg
};
P[2045]{
   GP1:
	UF : 0, UT : 6,		CONFIG : 'N U T, 0, 0, 0',
	X =  259.345  mm,	Y =   -346.085  mm,	Z =   -309.100  mm,
	W =  90.000 deg,	P =   0.000 deg,	R =   90.000 deg
};
P[2046]{
   GP1:
	UF : 0, UT : 6,		CONFIG : 'N U T, 0, 0, 0',
	X =  258.804  mm,	Y =   -346.894  mm,	Z =   -309.000  mm,
	W =  90.000 deg,	P =   0.000 deg,	R =   90.000 deg
};
P[2047]{
   GP1:
	UF : 0, UT : 6,		CONFIG : 'N U T, 0, 0, 0',
	X =  257.874  mm,	Y =   -347.471  mm,	Z =   -309.100  mm,
	W =  90.000 deg,	P =   0.000 deg,	R =   90.000 deg
};
P[2048]{
   GP1:
	UF : 0, UT : 6,		CONFIG : 'N U T, 0, 0, 0',
	X =  256.076  mm,	Y =   -348.533  mm,	Z =   -309.000  mm,
	W =  90.000 deg,	P =   0.000 deg,	R =   90.000 deg
};
P[2049]{
   GP1:
	UF : 0, UT : 6,		CONFIG : 'N U T, 0, 0, 0',
	X =  254.555  mm,	Y =   -348.969  mm,	Z =   -309.000  mm,
	W =  90.000 deg,	P =   0.000 deg,	R =   90.000 deg
};
P[2050]{
   GP1:
	UF : 0, UT : 6,		CONFIG : 'N U T, 0, 0, 0',
	X =  253.552  mm,	Y =   -349.604  mm,	Z =   -309.000  mm,
	W =  90.000 deg,	P =   0.000 deg,	R =   90.000 deg
};
P[2051]{
   GP1:
	UF : 0, UT : 6,		CONFIG : 'N U T, 0, 0, 0',
	X =  252.056  mm,	Y =   -350.443  mm,	Z =   -315.014  mm,
	W =  90.000 deg,	P =   0.000 deg,	R =   90.000 deg
};
P[2052]{
   GP1:
	UF : 0, UT : 6,		CONFIG : 'N U T, 0, 0, 0',
	X =  251.410  mm,	Y =   -350.933  mm,	Z =   -309.100  mm,
	W =  90.000 deg,	P =   0.000 deg,	R =   90.000 deg
};
P[2053]{
   GP1:
	UF : 0, UT : 6,		CONFIG : 'N U T, 0, 0, 0',
	X =  251.006  mm,	Y =   -351.536  mm,	Z =   -309.000  mm,
	W =  90.000 deg,	P =   0.000 deg,	R =   90.000 deg
};
P[2054]{
   GP1:
	UF : 0, UT : 6,		CONFIG : 'N U T, 0, 0, 0',
	X =  250.016  mm,	Y =   -351.876  mm,	Z =   -309.000  mm,
	W =  90.000 deg,	P =   0.000 deg,	R =   90.000 deg
};
P[2055]{
   GP1:
	UF : 0, UT : 6,		CONFIG : 'N U T, 0, 0, 0',
	X =  249.050  mm,	Y =   -352.442  mm,	Z =   -309.000  mm,
	W =  90.000 deg,	P =   0.000 deg,	R =   90.000 deg
};
P[2056]{
   GP1:
	UF : 0, UT : 6,		CONFIG : 'N U T, 0, 0, 0',
	X =  247.746  mm,	Y =   -352.980  mm,	Z =   -309.100  mm,
	W =  90.000 deg,	P =   0.000 deg,	R =   90.000 deg
};
P[2057]{
   GP1:
	UF : 0, UT : 6,		CONFIG : 'N U T, 0, 0, 0',
	X =  247.157  mm,	Y =   -353.704  mm,	Z =   -309.000  mm,
	W =  90.000 deg,	P =   0.000 deg,	R =   90.000 deg
};
P[2058]{
   GP1:
	UF : 0, UT : 6,		CONFIG : 'N U T, 0, 0, 0',
	X =  245.778  mm,	Y =   -354.070  mm,	Z =   -309.000  mm,
	W =  90.000 deg,	P =   0.000 deg,	R =   90.000 deg
};
P[2059]{
   GP1:
	UF : 0, UT : 6,		CONFIG : 'N U T, 0, 0, 0',
	X =  244.761  mm,	Y =   -355.239  mm,	Z =   -309.100  mm,
	W =  90.000 deg,	P =   0.000 deg,	R =   90.000 deg
};
P[2060]{
   GP1:
	UF : 0, UT : 6,		CONFIG : 'N U T, 0, 0, 0',
	X =  243.583  mm,	Y =   -356.018  mm,	Z =   -309.000  mm,
	W =  90.000 deg,	P =   0.000 deg,	R =   90.000 deg
};
P[2061]{
   GP1:
	UF : 0, UT : 6,		CONFIG : 'N U T, 0, 0, 0',
	X =  242.938  mm,	Y =   -356.466  mm,	Z =   -309.000  mm,
	W =  90.000 deg,	P =   0.000 deg,	R =   90.000 deg
};
P[2062]{
   GP1:
	UF : 0, UT : 6,		CONFIG : 'N U T, 0, 0, 0',
	X =  241.894  mm,	Y =   -356.361  mm,	Z =   -309.000  mm,
	W =  90.000 deg,	P =   0.000 deg,	R =   90.000 deg
};
P[2063]{
   GP1:
	UF : 0, UT : 6,		CONFIG : 'N U T, 0, 0, 0',
	X =  241.006  mm,	Y =   -357.306  mm,	Z =   -309.320  mm,
	W =  90.000 deg,	P =   0.000 deg,	R =   90.000 deg
};
P[2064]{
   GP1:
	UF : 0, UT : 6,		CONFIG : 'N U T, 0, 0, 0',
	X =  240.171  mm,	Y =   -357.895  mm,	Z =   -309.000  mm,
	W =  90.000 deg,	P =   0.000 deg,	R =   90.000 deg
};
P[2065]{
   GP1:
	UF : 0, UT : 6,		CONFIG : 'N U T, 0, 0, 0',
	X =  239.307  mm,	Y =   -358.241  mm,	Z =   -311.193  mm,
	W =  90.000 deg,	P =   0.000 deg,	R =   90.000 deg
};
P[2066]{
   GP1:
	UF : 0, UT : 6,		CONFIG : 'N U T, 0, 0, 0',
	X =  237.856  mm,	Y =   -358.790  mm,	Z =   -309.100  mm,
	W =  90.000 deg,	P =   0.000 deg,	R =   90.000 deg
};
P[2067]{
   GP1:
	UF : 0, UT : 6,		CONFIG : 'N U T, 0, 0, 0',
	X =  237.179  mm,	Y =   -359.242  mm,	Z =   -309.000  mm,
	W =  90.000 deg,	P =   0.000 deg,	R =   90.000 deg
};
P[2068]{
   GP1:
	UF : 0, UT : 6,		CONFIG : 'N U T, 0, 0, 0',
	X =  235.974  mm,	Y =   -359.921  mm,	Z =   -309.000  mm,
	W =  90.000 deg,	P =   0.000 deg,	R =   90.000 deg
};
P[2069]{
   GP1:
	UF : 0, UT : 6,		CONFIG : 'N U T, 0, 0, 0',
	X =  234.849  mm,	Y =   -360.540  mm,	Z =   -309.000  mm,
	W =  90.000 deg,	P =   0.000 deg,	R =   90.000 deg
};
P[2070]{
   GP1:
	UF : 0, UT : 6,		CONFIG : 'N U T, 0, 0, 0',
	X =  233.749  mm,	Y =   -360.981  mm,	Z =   -320.247  mm,
	W =  90.000 deg,	P =   0.000 deg,	R =   90.000 deg
};
P[2071]{
   GP1:
	UF : 0, UT : 6,		CONFIG : 'N U T, 0, 0, 0',
	X =  232.846  mm,	Y =   -361.735  mm,	Z =   -319.870  mm,
	W =  90.000 deg,	P =   0.000 deg,	R =   90.000 deg
};
P[2072]{
   GP1:
	UF : 0, UT : 6,		CONFIG : 'N U T, 0, 0, 0',
	X =  232.015  mm,	Y =   -362.623  mm,	Z =   -309.000  mm,
	W =  90.000 deg,	P =   0.000 deg,	R =   90.000 deg
};
P[2073]{
   GP1:
	UF : 0, UT : 6,		CONFIG : 'N U T, 0, 0, 0',
	X =  230.797  mm,	Y =   -362.624  mm,	Z =   -309.000  mm,
	W =  90.000 deg,	P =   0.000 deg,	R =   90.000 deg
};
P[2074]{
   GP1:
	UF : 0, UT : 6,		CONFIG : 'N U T, 0, 0, 0',
	X =  230.074  mm,	Y =   -363.705  mm,	Z =   -309.000  mm,
	W =  90.000 deg,	P =   0.000 deg,	R =   90.000 deg
};
P[2075]{
   GP1:
	UF : 0, UT : 6,		CONFIG : 'N U T, 0, 0, 0',
	X =  228.974  mm,	Y =   -364.438  mm,	Z =   -309.100  mm,
	W =  90.000 deg,	P =   0.000 deg,	R =   90.000 deg
};
P[2076]{
   GP1:
	UF : 0, UT : 6,		CONFIG : 'N U T, 0, 0, 0',
	X =  228.202  mm,	Y =   -364.705  mm,	Z =   -309.100  mm,
	W =  90.000 deg,	P =   0.000 deg,	R =   90.000 deg
};
P[2077]{
   GP1:
	UF : 0, UT : 6,		CONFIG : 'N U T, 0, 0, 0',
	X =  227.253  mm,	Y =   -364.685  mm,	Z =   -309.000  mm,
	W =  90.000 deg,	P =   0.000 deg,	R =   90.000 deg
};
P[2078]{
   GP1:
	UF : 0, UT : 6,		CONFIG : 'N U T, 0, 0, 0',
	X =  226.783  mm,	Y =   -365.697  mm,	Z =   -309.000  mm,
	W =  90.000 deg,	P =   0.000 deg,	R =   90.000 deg
};
P[2079]{
   GP1:
	UF : 0, UT : 6,		CONFIG : 'N U T, 0, 0, 0',
	X =  225.617  mm,	Y =   -365.962  mm,	Z =   -309.000  mm,
	W =  90.000 deg,	P =   0.000 deg,	R =   90.000 deg
};
P[2080]{
   GP1:
	UF : 0, UT : 6,		CONFIG : 'N U T, 0, 0, 0',
	X =  224.313  mm,	Y =   -366.419  mm,	Z =   -309.100  mm,
	W =  90.000 deg,	P =   0.000 deg,	R =   90.000 deg
};
P[2081]{
   GP1:
	UF : 0, UT : 6,		CONFIG : 'N U T, 0, 0, 0',
	X =  224.005  mm,	Y =   -367.349  mm,	Z =   -322.039  mm,
	W =  90.000 deg,	P =   0.000 deg,	R =   90.000 deg
};
P[2082]{
   GP1:
	UF : 0, UT : 6,		CONFIG : 'N U T, 0, 0, 0',
	X =  223.148  mm,	Y =   -367.303  mm,	Z =   -309.000  mm,
	W =  90.000 deg,	P =   0.000 deg,	R =   90.000 deg
};
P[2083]{
   GP1:
	UF : 0, UT : 6,		CONFIG : 'N U T, 0, 0, 0',
	X =  222.192  mm,	Y =   -368.204  mm,	Z =   -309.100  mm,
	W =  90.000 deg,	P =   0.000 deg,	R =   90.000 deg
};
P[2084]{
   GP1:
	UF : 0, UT : 6,		CONFIG : 'N U T, 0, 0, 0',
	X =  221.083  mm,	Y =   -368.693  mm,	Z =   -309.000  mm,
	W =  90.000 deg,	P =   0.000 deg,	R =   90.000 deg
};
P[2085]{
   GP1:
	UF : 0, UT : 6,		CONFIG : 'N U T, 0, 0, 0',
	X =  219.920  mm,	Y =   -369.296  mm,	Z =   -309.000  mm,
	W =  90.000 deg,	P =   0.000 deg,	R =   90.000 deg
};
P[2086]{
   GP1:
	UF : 0, UT : 6,		CONFIG : 'N U T, 0, 0, 0',
	X =  219.107  mm,	Y =   -369.932  mm,	Z =   -309.000  mm,
	W =  90.000 deg,	P =   0.000 deg,	R =   90.000 deg
};
P[2087]{
   GP1:
	UF : 0, UT : 6,		CONFIG : 'N U T, 0, 0, 0',
	X =  217.786  mm,	Y =   -370.291  mm,	Z =   -320.737  mm,
	W =  90.000 deg,	P =   0.000 deg,	R =   90.000 deg
};
P[2088]{
   GP1:
	UF : 0, UT : 6,		CONFIG : 'N U T, 0, 0, 0',
	X =  217.010  mm,	Y =   -370.849  mm,	Z =   -309.100  mm,
	W =  90.000 deg,	P =   0.000 deg,	R =   90.000 deg
};
P[2089]{
   GP1:
	UF : 0, UT : 6,		CONFIG : 'N U T, 0, 0, 0',
	X =  215.964  mm,	Y =   -371.517  mm,	Z =   -309.000  mm,
	W =  90.000 deg,	P =   0.000 deg,	R =   90.000 deg
};
P[2090]{
   GP1:
	UF : 0, UT : 6,		CONFIG : 'N U T, 0, 0, 0',
	X =  215.150  mm,	Y =   -372.482  mm,	Z =   -309.100  mm,
	W =  90.000 deg,	P =   0.000 deg,	R =   90.000 deg
};
P[2091]{
   GP1:
	UF : 0, UT : 6,		CONFIG : 'N U T, 0, 0, 0',
	X =  214.345  mm,	Y =   -372.373  mm,	Z =   -309.000  mm,
	W =  90.000 deg,	P =   0.000 deg,	R =   90.000 deg
};
P[2092]{
   GP1:
	UF : 0, UT : 6,		CONFIG : 'N U T, 0, 0, 0',
	X =  213.421  mm,	Y =   -373.565  mm,	Z =   -309.000  mm,
	W =  90.000 deg,	P =   0.000 deg,	R =   90.000 deg
};
P[2093]{
   GP1:
	UF : 0, UT : 6,		CONFIG : 'N U T, 0, 0, 0',
	X =  212.745  mm,	Y =   -373.274  mm,	Z =   -309.100  mm,
	W =  90.000 deg,	P =   0.000 deg,	R =   90.000 deg
};
P[2094]{
   GP1:
	UF : 0, UT : 6,		CONFIG : 'N U T, 0, 0, 0',
	X =  212.216  mm,	Y =   -373.983  mm,	Z =   -309.000  mm,
	W =  90.000 deg,	P =   0.000 deg,	R =   90.000 deg
};
P[2095]{
   GP1:
	UF : 0, UT : 6,		CONFIG : 'N U T, 0, 0, 0',
	X =  211.141  mm,	Y =   -374.511  mm,	Z =   -309.000  mm,
	W =  90.000 deg,	P =   0.000 deg,	R =   90.000 deg
};
P[2096]{
   GP1:
	UF : 0, UT : 6,		CONFIG : 'N U T, 0, 0, 0',
	X =  209.982  mm,	Y =   -374.811  mm,	Z =   -309.000  mm,
	W =  90.000 deg,	P =   0.000 deg,	R =   90.000 deg
};
P[2097]{
   GP1:
	UF : 0, UT : 6,		CONFIG : 'N U T, 0, 0, 0',
	X =  208.926  mm,	Y =   -375.486  mm,	Z =   -309.000  mm,
	W =  90.000 deg,	P =   0.000 deg,	R =   90.000 deg
};
P[2098]{
   GP1:
	UF : 0, UT : 6,		CONFIG : 'N U T, 0, 0, 0',
	X =  208.343  mm,	Y =   -376.128  mm,	Z =   -309.000  mm,
	W =  90.000 deg,	P =   0.000 deg,	R =   90.000 deg
};
P[2099]{
   GP1:
	UF : 0, UT : 6,		CONFIG : 'N U T, 0, 0, 0',
	X =  207.163  mm,	Y =   -376.694  mm,	Z =   -309.000  mm,
	W =  90.000 deg,	P =   0.000 deg,	R =   90.000 deg
};
P[2100]{
   GP1:
	UF : 0, UT : 6,		CONFIG : 'N U T, 0, 0, 0',
	X =  206.417  mm,	Y =   -376.708  mm,	Z =   -311.352  mm,
	W =  90.000 deg,	P =   0.000 deg,	R =   90.000 deg
};
P[2101]{
   GP1:
	UF : 0, UT : 6,		CONFIG : 'N U T, 0, 0, 0',
	X =  205.107  mm,	Y =   -378.324  mm,	Z =   -309.100  mm,
	W =  90.000 deg,	P =   0.000 deg,	R =   90.000 deg
};
P[2102]{
   GP1:
	UF : 0, UT : 6,		CONFIG : 'N U T, 0, 0, 0',
	X =  204.134  mm,	Y =   -378.436  mm,	Z =   -309.000  mm,
	W =  90.000 deg,	P =   0.000 deg,	R =   90.000 deg
};
P[2103]{
   GP1:
	UF : 0, UT : 6,		CONFIG : 'N U T, 0, 0, 0',
	X =  203.340  mm,	Y =   -379.412  mm,	Z =   -309.000  mm,
	W =  90.000 deg,	P =   0.000 deg,	R =   90.000 deg
};
P[2104]{
   GP1:
	UF : 0, UT : 6,		CONFIG : 'N U T, 0, 0, 0',
	X =  202.543  mm,	Y =   -379.372  mm,	Z =   -309.000  mm,
	W =  90.000 deg,	P =   0.000 deg,	R =   90.000 deg
};
P[2105]{
   GP1:
	UF : 0, UT : 6,		CONFIG : 'N U T, 0, 0, 0',
	X =  201.478  mm,	Y =   -380.168  mm,	Z =   -309.100  mm,
	W =  90.000 deg,	P =   0.000 deg,	R =   90.000 deg
};
P[2106]{
   GP1:
	UF : 0, UT : 6,		CONFIG : 'N U T, 0, 0, 0',
	X =  200.489  mm,	Y =   -380.068  mm,	Z =   -309.000  mm,
	W =  90.000 deg,	P =   0.000 deg,	R =   90.000 deg
};
P[2107]{
   GP1:
	UF : 0, UT : 6,		CONFIG : 'N U T, 0, 0, 0',
	X =  199.539  mm,	Y =   -381.171  mm,	Z =   -309.000  mm,
	W =  90.000 deg,	P =   0.000 deg,	R =   90.000 deg
};
P[2108]{
   GP1:
	UF : 0, UT : 6,		CONFIG : 'N U T, 0, 0, 0',
	X =  198.727  mm,	Y =   -381.687  mm,	Z =   -309.000  mm,
	W =  90.000 deg,	P =   0.000 deg,	R =   90.000 deg
};
P[2109]{
   GP1:
	UF : 0, UT : 6,		CONFIG : 'N U T, 0, 0, 0',
	X =  197.885  mm,	Y =   -381.430  mm,	Z =   -321.626  mm,
	W =  90.000 deg,	P =   0.000 deg,	R =   90.000 deg
};
P[2110]{
   GP1:
	UF : 0, UT : 6,		CONFIG : 'N U T, 0, 0, 0',
	X =  196.949  mm,	Y =   -382.352  mm,	Z =   -309.000  mm,
	W =  90.000 deg,	P =   0.000 deg,	R =   90.000 deg
};
P[2111]{
   GP1:
	UF : 0, UT : 6,		CONFIG : 'N U T, 0, 0, 0',
	X =  196.103  mm,	Y =   -382.750  mm,	Z =   -309.000  mm,
	W =  90.000 deg,	P =   0.000 deg,	R =   90.000 deg
};
P[2112]{
   GP1:
	UF : 0, UT : 6,		CONFIG : 'N U T, 0, 0, 0',
	X =  195.291  mm,	Y =   -383.293  mm,	Z =   -309.100  mm,
	W =  90.000 deg,	P =   0.000 deg,	R =   90.000 deg
};
P[2113]{
   GP1:
	UF : 0, UT : 6,		CONFIG : 'N U T, 0, 0, 0',
	X =  194.670  mm,	Y =   -383.774  mm,	Z =   -314.345  mm,
	W =  90.000 deg,	P =   0.000 deg,	R =   90.000 deg
};
P[2114]{
   GP1:
	UF : 0, UT : 6,		CONFIG : 'N U T, 0, 0, 0',
	X =  193.439  mm,	Y =   -384.516  mm,	Z =   -309.000  mm,
	W =  90.000 deg,	P =   0.000 deg,	R =   90.000 deg
};
P[2115]{
   GP1:
	UF : 0, UT : 6,		CONFIG : 'N U T, 0, 0, 0',
	X =  191.668  mm,	Y =   -385.662  mm,	Z =   -309.000  mm,
	W =  90.000 deg,	P =   0.000 deg,	R =   90.000 deg
};
P[2116]{
   GP1:
	UF : 0, UT : 6,		CONFIG : 'N U T, 0, 0, 0',
	X =  190.617  mm,	Y =   -385.726  mm,	Z =   -309.000  mm,
	W =  90.000 deg,	P =   0.000 deg,	R =   90.000 deg
};
P[2117]{
   GP1:
	UF : 0, UT : 6,		CONFIG : 'N U T, 0, 0, 0',
	X =  189.920  mm,	Y =   -386.383  mm,	Z =   -309.000  mm,
	W =  90.000 deg,	P =   0.000 deg,	R =   90.000 deg
};
P[2118]{
   GP1:
	UF : 0, UT : 6,		CONFIG : 'N U T, 0, 0, 0',
	X =  189.185  mm,	Y =   -386.772  mm,	Z =   -309.100  mm,
	W =  90.000 deg,	P =   0.000 deg,	R =   90.000 deg
};
P[2119]{
   GP1:
	UF : 0, UT : 6,		CONFIG : 'N U T, 0, 0, 0',
	X =  188.211  mm,	Y =   -387.117  mm,	Z =   -322.286  mm,
	W =  90.000 deg,	P =   0.000 deg,	R =   90.000 deg
};
P[2120]{
   GP1:
	UF : 0, UT : 6,		CONFIG : 'N U T, 0, 0, 0',
	X =  187.636  mm,	Y =   -388.248  mm,	Z =   -320.295  mm,
	W =  90.000 deg,	P =   0.000 deg,	R =   90.000 deg
};
P[2121]{
   GP1:
	UF : 0, UT : 6,		CONFIG : 'N U T, 0, 0, 0',
	X =  186.334  mm,	Y =   -388.419  mm,	Z =   -309.100  mm,
	W =  90.000 deg,	P =   0.000 deg,	R =   90.000 deg
};
P[2122]{
   GP1:
	UF : 0, UT : 6,		CONFIG : 'N U T, 0, 0, 0',
	X =  185.585  mm,	Y =   -389.059  mm,	Z =   -311.564  mm,
	W =  90.000 deg,	P =   0.000 deg,	R =   90.000 deg
};
P[2123]{
   GP1:
	UF : 0, UT : 6,		CONFIG : 'N U T, 0, 0, 0',
	X =  185.188  mm,	Y =   -389.856  mm,	Z =   -309.000  mm,
	W =  90.000 deg,	P =   0.000 deg,	R =   90.000 deg
};
P[2124]{
   GP1:
	UF : 0, UT : 6,		CONFIG : 'N U T, 0, 0, 0',
	X =  184.063  mm,	Y =   -389.918  mm,	Z =   -309.000  mm,
	W =  90.000 deg,	P =   0.000 deg,	R =   90.000 deg
};
P[2125]{
   GP1:
	UF : 0, UT : 6,		CONFIG : 'N U T, 0, 0, 0',
	X =  183.308  mm,	Y =   -390.980  mm,	Z =   -309.000  mm,
	W =  90.000 deg,	P =   0.000 deg,	R =   90.000 deg
};
P[2126]{
   GP1:
	UF : 0, UT : 6,		CONFIG : 'N U T, 0, 0, 0',
	X =  181.909  mm,	Y =   -390.825  mm,	Z =   -309.000  mm,
	W =  90.000 deg,	P =   0.000 deg,	R =   90.000 deg
};
P[2127]{
   GP1:
	UF : 0, UT : 6,		CONFIG : 'N U T, 0, 0, 0',
	X =  181.503  mm,	Y =   -391.445  mm,	Z =   -309.000  mm,
	W =  90.000 deg,	P =   0.000 deg,	R =   90.000 deg
};
P[2128]{
   GP1:
	UF : 0, UT : 6,		CONFIG : 'N U T, 0, 0, 0',
	X =  180.908  mm,	Y =   -391.947  mm,	Z =   -309.000  mm,
	W =  90.000 deg,	P =   0.000 deg,	R =   90.000 deg
};
P[2129]{
   GP1:
	UF : 0, UT : 6,		CONFIG : 'N U T, 0, 0, 0',
	X =  179.787  mm,	Y =   -392.278  mm,	Z =   -309.100  mm,
	W =  90.000 deg,	P =   0.000 deg,	R =   90.000 deg
};
P[2130]{
   GP1:
	UF : 0, UT : 6,		CONFIG : 'N U T, 0, 0, 0',
	X =  179.065  mm,	Y =   -392.859  mm,	Z =   -309.000  mm,
	W =  90.000 deg,	P =   0.000 deg,	R =   90.000 deg
};
P[2131]{
   GP1:
	UF : 0, UT : 6,		CONFIG : 'N U T, 0, 0, 0',
	X =  178.041  mm,	Y =   -392.984  mm,	Z =   -309.000  mm,
	W =  90.000 deg,	P =   0.000 deg,	R =   90.000 deg
};
P[2132]{
   GP1:
	UF : 0, UT : 6,		CONFIG : 'N U T, 0, 0, 0',
	X =  177.280  mm,	Y =   -394.405  mm,	Z =   -309.000  mm,
	W =  90.000 deg,	P =   0.000 deg,	R =   90.000 deg
};
P[2133]{
   GP1:
	UF : 0, UT : 6,		CONFIG : 'N U T, 0, 0, 0',
	X =  176.564  mm,	Y =   -394.105  mm,	Z =   -309.100  mm,
	W =  90.000 deg,	P =   0.000 deg,	R =   90.000 deg
};
P[2134]{
   GP1:
	UF : 0, UT : 6,		CONFIG : 'N U T, 0, 0, 0',
	X =  175.782  mm,	Y =   -394.809  mm,	Z =   -309.000  mm,
	W =  90.000 deg,	P =   0.000 deg,	R =   90.000 deg
};
P[2135]{
   GP1:
	UF : 0, UT : 6,		CONFIG : 'N U T, 0, 0, 0',
	X =  174.424  mm,	Y =   -395.435  mm,	Z =   -309.000  mm,
	W =  90.000 deg,	P =   0.000 deg,	R =   90.000 deg
};
P[2136]{
   GP1:
	UF : 0, UT : 6,		CONFIG : 'N U T, 0, 0, 0',
	X =  173.660  mm,	Y =   -395.973  mm,	Z =   -309.000  mm,
	W =  90.000 deg,	P =   0.000 deg,	R =   90.000 deg
};
P[2137]{
   GP1:
	UF : 0, UT : 6,		CONFIG : 'N U T, 0, 0, 0',
	X =  172.757  mm,	Y =   -396.304  mm,	Z =   -309.100  mm,
	W =  90.000 deg,	P =   0.000 deg,	R =   90.000 deg
};
P[2138]{
   GP1:
	UF : 0, UT : 6,		CONFIG : 'N U T, 0, 0, 0',
	X =  171.940  mm,	Y =   -397.060  mm,	Z =   -309.000  mm,
	W =  90.000 deg,	P =   0.000 deg,	R =   90.000 deg
};
P[2139]{
   GP1:
	UF : 0, UT : 6,		CONFIG : 'N U T, 0, 0, 0',
	X =  170.331  mm,	Y =   -397.922  mm,	Z =   -309.000  mm,
	W =  90.000 deg,	P =   0.000 deg,	R =   90.000 deg
};
P[2140]{
   GP1:
	UF : 0, UT : 6,		CONFIG : 'N U T, 0, 0, 0',
	X =  169.354  mm,	Y =   -398.524  mm,	Z =   -309.000  mm,
	W =  90.000 deg,	P =   0.000 deg,	R =   90.000 deg
};
P[2141]{
   GP1:
	UF : 0, UT : 6,		CONFIG : 'N U T, 0, 0, 0',
	X =  168.171  mm,	Y =   -399.080  mm,	Z =   -309.000  mm,
	W =  90.000 deg,	P =   0.000 deg,	R =   90.000 deg
};
P[2142]{
   GP1:
	UF : 0, UT : 6,		CONFIG : 'N U T, 0, 0, 0',
	X =  166.706  mm,	Y =   -399.953  mm,	Z =   -309.000  mm,
	W =  90.000 deg,	P =   0.000 deg,	R =   90.000 deg
};
P[2143]{
   GP1:
	UF : 0, UT : 6,		CONFIG : 'N U T, 0, 0, 0',
	X =  165.577  mm,	Y =   -400.295  mm,	Z =   -327.655  mm,
	W =  90.000 deg,	P =   0.000 deg,	R =   90.000 deg
};
P[2144]{
   GP1:
	UF : 0, UT : 6,		CONFIG : 'N U T, 0, 0, 0',
	X =  164.907  mm,	Y =   -401.141  mm,	Z =   -309.000  mm,
	W =  90.000 deg,	P =   0.000 deg,	R =   90.000 deg
};
P[2145]{
   GP1:
	UF : 0, UT : 6,		CONFIG : 'N U T, 0, 0, 0',
	X =  164.071  mm,	Y =   -401.621  mm,	Z =   -326.631  mm,
	W =  90.000 deg,	P =   0.000 deg,	R =   90.000 deg
};
P[2146]{
   GP1:
	UF : 0, UT : 6,		CONFIG : 'N U T, 0, 0, 0',
	X =  163.027  mm,	Y =   -401.908  mm,	Z =   -309.000  mm,
	W =  90.000 deg,	P =   0.000 deg,	R =   90.000 deg
};
P[2147]{
   GP1:
	UF : 0, UT : 6,		CONFIG : 'N U T, 0, 0, 0',
	X =  162.168  mm,	Y =   -402.713  mm,	Z =   -317.253  mm,
	W =  90.000 deg,	P =   0.000 deg,	R =   90.000 deg
};
P[2148]{
   GP1:
	UF : 0, UT : 6,		CONFIG : 'N U T, 0, 0, 0',
	X =  161.602  mm,	Y =   -403.457  mm,	Z =   -309.000  mm,
	W =  90.000 deg,	P =   0.000 deg,	R =   90.000 deg
};
P[2149]{
   GP1:
	UF : 0, UT : 6,		CONFIG : 'N U T, 0, 0, 0',
	X =  160.647  mm,	Y =   -403.436  mm,	Z =   -309.100  mm,
	W =  90.000 deg,	P =   0.000 deg,	R =   90.000 deg
};
P[2150]{
   GP1:
	UF : 0, UT : 6,		CONFIG : 'N U T, 0, 0, 0',
	X =  159.650  mm,	Y =   -404.617  mm,	Z =   -316.578  mm,
	W =  90.000 deg,	P =   0.000 deg,	R =   90.000 deg
};
P[2151]{
   GP1:
	UF : 0, UT : 6,		CONFIG : 'N U T, 0, 0, 0',
	X =  158.608  mm,	Y =   -404.631  mm,	Z =   -314.391  mm,
	W =  90.000 deg,	P =   0.000 deg,	R =   90.000 deg
};
P[2152]{
   GP1:
	UF : 0, UT : 6,		CONFIG : 'N U T, 0, 0, 0',
	X =  157.505  mm,	Y =   -404.907  mm,	Z =   -318.908  mm,
	W =  90.000 deg,	P =   0.000 deg,	R =   90.000 deg
};
P[2153]{
   GP1:
	UF : 0, UT : 6,		CONFIG : 'N U T, 0, 0, 0',
	X =  156.981  mm,	Y =   -405.461  mm,	Z =   -309.100  mm,
	W =  90.000 deg,	P =   0.000 deg,	R =   90.000 deg
};
P[2154]{
   GP1:
	UF : 0, UT : 6,		CONFIG : 'N U T, 0, 0, 0',
	X =  155.421  mm,	Y =   -406.380  mm,	Z =   -309.000  mm,
	W =  90.000 deg,	P =   0.000 deg,	R =   90.000 deg
};
P[2155]{
   GP1:
	UF : 0, UT : 6,		CONFIG : 'N U T, 0, 0, 0',
	X =  154.176  mm,	Y =   -406.849  mm,	Z =   -309.000  mm,
	W =  90.000 deg,	P =   0.000 deg,	R =   90.000 deg
};
P[2156]{
   GP1:
	UF : 0, UT : 6,		CONFIG : 'N U T, 0, 0, 0',
	X =  154.217  mm,	Y =   -407.606  mm,	Z =   -309.000  mm,
	W =  90.000 deg,	P =   0.000 deg,	R =   90.000 deg
};
P[2157]{
   GP1:
	UF : 0, UT : 6,		CONFIG : 'N U T, 0, 0, 0',
	X =  152.738  mm,	Y =   -407.908  mm,	Z =   -309.000  mm,
	W =  90.000 deg,	P =   0.000 deg,	R =   90.000 deg
};
P[2158]{
   GP1:
	UF : 0, UT : 6,		CONFIG : 'N U T, 0, 0, 0',
	X =  151.488  mm,	Y =   -408.642  mm,	Z =   -325.352  mm,
	W =  90.000 deg,	P =   0.000 deg,	R =   90.000 deg
};
P[2159]{
   GP1:
	UF : 0, UT : 6,		CONFIG : 'N U T, 0, 0, 0',
	X =  150.691  mm,	Y =   -408.822  mm,	Z =   -319.247  mm,
	W =  90.000 deg,	P =   0.000 deg,	R =   90.000 deg
};
P[2160]{
   GP1:
	UF : 0, UT : 6,		CONFIG : 'N U T, 0, 0, 0',
	X =  150.288  mm,	Y =   -409.609  mm,	Z =   -309.000  mm,
	W =  90.000 deg,	P =   0.000 deg,	R =   90.000 deg
};
P[2161]{
   GP1:
	UF : 0, UT : 6,		CONFIG : 'N U T, 0, 0, 0',
	X =  149.449  mm,	Y =   -409.876  mm,	Z =   -309.100  mm,
	W =  90.000 deg,	P =   0.000 deg,	R =   90.000 deg
};
P[2162]{
   GP1:
	UF : 0, UT : 6,		CONFIG : 'N U T, 0, 0, 0',
	X =  148.548  mm,	Y =   -410.562  mm,	Z =   -309.000  mm,
	W =  90.000 deg,	P =   0.000 deg,	R =   90.000 deg
};
P[2163]{
   GP1:
	UF : 0, UT : 6,		CONFIG : 'N U T, 0, 0, 0',
	X =  147.196  mm,	Y =   -410.866  mm,	Z =   -309.000  mm,
	W =  90.000 deg,	P =   0.000 deg,	R =   90.000 deg
};
P[2164]{
   GP1:
	UF : 0, UT : 6,		CONFIG : 'N U T, 0, 0, 0',
	X =  146.603  mm,	Y =   -411.600  mm,	Z =   -309.000  mm,
	W =  90.000 deg,	P =   0.000 deg,	R =   90.000 deg
};
P[2165]{
   GP1:
	UF : 0, UT : 6,		CONFIG : 'N U T, 0, 0, 0',
	X =  145.559  mm,	Y =   -412.103  mm,	Z =   -309.000  mm,
	W =  90.000 deg,	P =   0.000 deg,	R =   90.000 deg
};
P[2166]{
   GP1:
	UF : 0, UT : 6,		CONFIG : 'N U T, 0, 0, 0',
	X =  145.169  mm,	Y =   -412.724  mm,	Z =   -316.308  mm,
	W =  90.000 deg,	P =   0.000 deg,	R =   90.000 deg
};
P[2167]{
   GP1:
	UF : 0, UT : 6,		CONFIG : 'N U T, 0, 0, 0',
	X =  144.110  mm,	Y =   -413.209  mm,	Z =   -309.000  mm,
	W =  90.000 deg,	P =   0.000 deg,	R =   90.000 deg
};
P[2168]{
   GP1:
	UF : 0, UT : 6,		CONFIG : 'N U T, 0, 0, 0',
	X =  142.250  mm,	Y =   -413.922  mm,	Z =   -309.000  mm,
	W =  90.000 deg,	P =   0.000 deg,	R =   90.000 deg
};
P[2169]{
   GP1:
	UF : 0, UT : 6,		CONFIG : 'N U T, 0, 0, 0',
	X =  141.455  mm,	Y =   -414.419  mm,	Z =   -309.100  mm,
	W =  90.000 deg,	P =   0.000 deg,	R =   90.000 deg
};
P[2170]{
   GP1:
	UF : 0, UT : 6,		CONFIG : 'N U T, 0, 0, 0',
	X =  140.470  mm,	Y =   -414.897  mm,	Z =   -309.000  mm,
	W =  90.000 deg,	P =   0.000 deg,	R =   90.000 deg
};
P[2171]{
   GP1:
	UF : 0, UT : 6,		CONFIG : 'N U T, 0, 0, 0',
	X =  139.287  mm,	Y =   -415.899  mm,	Z =   -309.000  mm,
	W =  90.000 deg,	P =   0.000 deg,	R =   90.000 deg
};
P[2172]{
   GP1:
	UF : 0, UT : 6,		CONFIG : 'N U T, 0, 0, 0',
	X =  138.058  mm,	Y =   -416.573  mm,	Z =   -309.000  mm,
	W =  90.000 deg,	P =   0.000 deg,	R =   90.000 deg
};
P[2173]{
   GP1:
	UF : 0, UT : 6,		CONFIG : 'N U T, 0, 0, 0',
	X =  137.256  mm,	Y =   -417.064  mm,	Z =   -309.000  mm,
	W =  90.000 deg,	P =   0.000 deg,	R =   90.000 deg
};
P[2174]{
   GP1:
	UF : 0, UT : 6,		CONFIG : 'N U T, 0, 0, 0',
	X =  136.452  mm,	Y =   -417.346  mm,	Z =   -309.100  mm,
	W =  90.000 deg,	P =   0.000 deg,	R =   90.000 deg
};
P[2175]{
   GP1:
	UF : 0, UT : 6,		CONFIG : 'N U T, 0, 0, 0',
	X =  135.527  mm,	Y =   -418.577  mm,	Z =   -309.100  mm,
	W =  90.000 deg,	P =   0.000 deg,	R =   90.000 deg
};
P[2176]{
   GP1:
	UF : 0, UT : 6,		CONFIG : 'N U T, 0, 0, 0',
	X =  133.827  mm,	Y =   -418.969  mm,	Z =   -309.756  mm,
	W =  90.000 deg,	P =   0.000 deg,	R =   90.000 deg
};
P[2177]{
   GP1:
	UF : 0, UT : 6,		CONFIG : 'N U T, 0, 0, 0',
	X =  133.141  mm,	Y =   -419.853  mm,	Z =   -309.000  mm,
	W =  90.000 deg,	P =   0.000 deg,	R =   90.000 deg
};
P[2178]{
   GP1:
	UF : 0, UT : 6,		CONFIG : 'N U T, 0, 0, 0',
	X =  131.985  mm,	Y =   -419.954  mm,	Z =   -309.000  mm,
	W =  90.000 deg,	P =   0.000 deg,	R =   90.000 deg
};
P[2179]{
   GP1:
	UF : 0, UT : 6,		CONFIG : 'N U T, 0, 0, 0',
	X =  130.927  mm,	Y =   -420.751  mm,	Z =   -309.000  mm,
	W =  90.000 deg,	P =   0.000 deg,	R =   90.000 deg
};
P[2180]{
   GP1:
	UF : 0, UT : 6,		CONFIG : 'N U T, 0, 0, 0',
	X =  130.032  mm,	Y =   -421.313  mm,	Z =   -309.000  mm,
	W =  90.000 deg,	P =   0.000 deg,	R =   90.000 deg
};
P[2181]{
   GP1:
	UF : 0, UT : 6,		CONFIG : 'N U T, 0, 0, 0',
	X =  128.874  mm,	Y =   -421.806  mm,	Z =   -309.000  mm,
	W =  90.000 deg,	P =   0.000 deg,	R =   90.000 deg
};
P[2182]{
   GP1:
	UF : 0, UT : 6,		CONFIG : 'N U T, 0, 0, 0',
	X =  127.741  mm,	Y =   -422.460  mm,	Z =   -309.000  mm,
	W =  90.000 deg,	P =   0.000 deg,	R =   90.000 deg
};
P[2183]{
   GP1:
	UF : 0, UT : 6,		CONFIG : 'N U T, 0, 0, 0',
	X =  126.941  mm,	Y =   -422.966  mm,	Z =   -309.000  mm,
	W =  90.000 deg,	P =   0.000 deg,	R =   90.000 deg
};
P[2184]{
   GP1:
	UF : 0, UT : 6,		CONFIG : 'N U T, 0, 0, 0',
	X =  126.500  mm,	Y =   -423.597  mm,	Z =   -320.410  mm,
	W =  90.000 deg,	P =   0.000 deg,	R =   90.000 deg
};
P[2185]{
   GP1:
	UF : 0, UT : 6,		CONFIG : 'N U T, 0, 0, 0',
	X =  125.489  mm,	Y =   -423.760  mm,	Z =   -309.000  mm,
	W =  90.000 deg,	P =   0.000 deg,	R =   90.000 deg
};
P[2186]{
   GP1:
	UF : 0, UT : 6,		CONFIG : 'N U T, 0, 0, 0',
	X =  124.510  mm,	Y =   -424.576  mm,	Z =   -309.000  mm,
	W =  90.000 deg,	P =   0.000 deg,	R =   90.000 deg
};
P[2187]{
   GP1:
	UF : 0, UT : 6,		CONFIG : 'N U T, 0, 0, 0',
	X =  123.720  mm,	Y =   -425.300  mm,	Z =   -309.100  mm,
	W =  90.000 deg,	P =   0.000 deg,	R =   90.000 deg
};
P[2188]{
   GP1:
	UF : 0, UT : 6,		CONFIG : 'N U T, 0, 0, 0',
	X =  130.889  mm,	Y =   -437.879  mm,	Z =   -309.100  mm,
	W =  90.000 deg,	P =   0.000 deg,	R =   90.000 deg
};
P[2189]{
   GP1:
	UF : 0, UT : 6,		CONFIG : 'N U T, 0, 0, 0',
	X =  131.754  mm,	Y =   -437.377  mm,	Z =   -309.100  mm,
	W =  90.000 deg,	P =   0.000 deg,	R =   90.000 deg
};
P[2190]{
   GP1:
	UF : 0, UT : 6,		CONFIG : 'N U T, 0, 0, 0',
	X =  132.367  mm,	Y =   -436.642  mm,	Z =   -309.000  mm,
	W =  90.000 deg,	P =   0.000 deg,	R =   90.000 deg
};
P[2191]{
   GP1:
	UF : 0, UT : 6,		CONFIG : 'N U T, 0, 0, 0',
	X =  133.424  mm,	Y =   -436.740  mm,	Z =   -309.000  mm,
	W =  90.000 deg,	P =   0.000 deg,	R =   90.000 deg
};
P[2192]{
   GP1:
	UF : 0, UT : 6,		CONFIG : 'N U T, 0, 0, 0',
	X =  134.037  mm,	Y =   -436.286  mm,	Z =   -309.000  mm,
	W =  90.000 deg,	P =   0.000 deg,	R =   90.000 deg
};
P[2193]{
   GP1:
	UF : 0, UT : 6,		CONFIG : 'N U T, 0, 0, 0',
	X =  135.185  mm,	Y =   -436.024  mm,	Z =   -309.000  mm,
	W =  90.000 deg,	P =   0.000 deg,	R =   90.000 deg
};
P[2194]{
   GP1:
	UF : 0, UT : 6,		CONFIG : 'N U T, 0, 0, 0',
	X =  135.842  mm,	Y =   -435.356  mm,	Z =   -309.000  mm,
	W =  90.000 deg,	P =   0.000 deg,	R =   90.000 deg
};
P[2195]{
   GP1:
	UF : 0, UT : 6,		CONFIG : 'N U T, 0, 0, 0',
	X =  136.475  mm,	Y =   -434.572  mm,	Z =   -319.927  mm,
	W =  90.000 deg,	P =   0.000 deg,	R =   90.000 deg
};
P[2196]{
   GP1:
	UF : 0, UT : 6,		CONFIG : 'N U T, 0, 0, 0',
	X =  137.526  mm,	Y =   -434.336  mm,	Z =   -309.000  mm,
	W =  90.000 deg,	P =   0.000 deg,	R =   90.000 deg
};
P[2197]{
   GP1:
	UF : 0, UT : 6,		CONFIG : 'N U T, 0, 0, 0',
	X =  138.505  mm,	Y =   -433.345  mm,	Z =   -309.000  mm,
	W =  90.000 deg,	P =   0.000 deg,	R =   90.000 deg
};
P[2198]{
   GP1:
	UF : 0, UT : 6,		CONFIG : 'N U T, 0, 0, 0',
	X =  139.248  mm,	Y =   -432.667  mm,	Z =   -309.000  mm,
	W =  90.000 deg,	P =   0.000 deg,	R =   90.000 deg
};
P[2199]{
   GP1:
	UF : 0, UT : 6,		CONFIG : 'N U T, 0, 0, 0',
	X =  140.280  mm,	Y =   -433.127  mm,	Z =   -314.260  mm,
	W =  90.000 deg,	P =   0.000 deg,	R =   90.000 deg
};
P[2200]{
   GP1:
	UF : 0, UT : 6,		CONFIG : 'N U T, 0, 0, 0',
	X =  141.681  mm,	Y =   -432.106  mm,	Z =   -309.100  mm,
	W =  90.000 deg,	P =   0.000 deg,	R =   90.000 deg
};
P[2201]{
   GP1:
	UF : 0, UT : 6,		CONFIG : 'N U T, 0, 0, 0',
	X =  142.123  mm,	Y =   -431.467  mm,	Z =   -309.000  mm,
	W =  90.000 deg,	P =   0.000 deg,	R =   90.000 deg
};
P[2202]{
   GP1:
	UF : 0, UT : 6,		CONFIG : 'N U T, 0, 0, 0',
	X =  143.065  mm,	Y =   -430.796  mm,	Z =   -309.000  mm,
	W =  90.000 deg,	P =   0.000 deg,	R =   90.000 deg
};
P[2203]{
   GP1:
	UF : 0, UT : 6,		CONFIG : 'N U T, 0, 0, 0',
	X =  144.227  mm,	Y =   -429.890  mm,	Z =   -309.100  mm,
	W =  90.000 deg,	P =   0.000 deg,	R =   90.000 deg
};
P[2204]{
   GP1:
	UF : 0, UT : 6,		CONFIG : 'N U T, 0, 0, 0',
	X =  145.390  mm,	Y =   -429.889  mm,	Z =   -314.091  mm,
	W =  90.000 deg,	P =   0.000 deg,	R =   90.000 deg
};
P[2205]{
   GP1:
	UF : 0, UT : 6,		CONFIG : 'N U T, 0, 0, 0',
	X =  146.419  mm,	Y =   -429.084  mm,	Z =   -309.000  mm,
	W =  90.000 deg,	P =   0.000 deg,	R =   90.000 deg
};
P[2206]{
   GP1:
	UF : 0, UT : 6,		CONFIG : 'N U T, 0, 0, 0',
	X =  147.506  mm,	Y =   -428.394  mm,	Z =   -309.000  mm,
	W =  90.000 deg,	P =   0.000 deg,	R =   90.000 deg
};
P[2207]{
   GP1:
	UF : 0, UT : 6,		CONFIG : 'N U T, 0, 0, 0',
	X =  149.071  mm,	Y =   -427.431  mm,	Z =   -309.100  mm,
	W =  90.000 deg,	P =   0.000 deg,	R =   90.000 deg
};
P[2208]{
   GP1:
	UF : 0, UT : 6,		CONFIG : 'N U T, 0, 0, 0',
	X =  150.189  mm,	Y =   -426.575  mm,	Z =   -309.000  mm,
	W =  90.000 deg,	P =   0.000 deg,	R =   90.000 deg
};
P[2209]{
   GP1:
	UF : 0, UT : 6,		CONFIG : 'N U T, 0, 0, 0',
	X =  151.643  mm,	Y =   -425.751  mm,	Z =   -309.000  mm,
	W =  90.000 deg,	P =   0.000 deg,	R =   90.000 deg
};
P[2210]{
   GP1:
	UF : 0, UT : 6,		CONFIG : 'N U T, 0, 0, 0',
	X =  152.447  mm,	Y =   -425.508  mm,	Z =   -309.100  mm,
	W =  90.000 deg,	P =   0.000 deg,	R =   90.000 deg
};
P[2211]{
   GP1:
	UF : 0, UT : 6,		CONFIG : 'N U T, 0, 0, 0',
	X =  153.296  mm,	Y =   -424.830  mm,	Z =   -309.100  mm,
	W =  90.000 deg,	P =   0.000 deg,	R =   90.000 deg
};
P[2212]{
   GP1:
	UF : 0, UT : 6,		CONFIG : 'N U T, 0, 0, 0',
	X =  154.570  mm,	Y =   -424.624  mm,	Z =   -309.100  mm,
	W =  90.000 deg,	P =   0.000 deg,	R =   90.000 deg
};
P[2213]{
   GP1:
	UF : 0, UT : 6,		CONFIG : 'N U T, 0, 0, 0',
	X =  155.909  mm,	Y =   -423.579  mm,	Z =   -309.100  mm,
	W =  90.000 deg,	P =   0.000 deg,	R =   90.000 deg
};
P[2214]{
   GP1:
	UF : 0, UT : 6,		CONFIG : 'N U T, 0, 0, 0',
	X =  156.920  mm,	Y =   -423.248  mm,	Z =   -309.000  mm,
	W =  90.000 deg,	P =   0.000 deg,	R =   90.000 deg
};
P[2215]{
   GP1:
	UF : 0, UT : 6,		CONFIG : 'N U T, 0, 0, 0',
	X =  157.646  mm,	Y =   -422.686  mm,	Z =   -309.000  mm,
	W =  90.000 deg,	P =   0.000 deg,	R =   90.000 deg
};
P[2216]{
   GP1:
	UF : 0, UT : 6,		CONFIG : 'N U T, 0, 0, 0',
	X =  158.549  mm,	Y =   -421.554  mm,	Z =   -309.000  mm,
	W =  90.000 deg,	P =   0.000 deg,	R =   90.000 deg
};
P[2217]{
   GP1:
	UF : 0, UT : 6,		CONFIG : 'N U T, 0, 0, 0',
	X =  159.733  mm,	Y =   -421.816  mm,	Z =   -309.100  mm,
	W =  90.000 deg,	P =   0.000 deg,	R =   90.000 deg
};
P[2218]{
   GP1:
	UF : 0, UT : 6,		CONFIG : 'N U T, 0, 0, 0',
	X =  160.677  mm,	Y =   -421.057  mm,	Z =   -309.000  mm,
	W =  90.000 deg,	P =   0.000 deg,	R =   90.000 deg
};
P[2219]{
   GP1:
	UF : 0, UT : 6,		CONFIG : 'N U T, 0, 0, 0',
	X =  161.261  mm,	Y =   -420.596  mm,	Z =   -309.000  mm,
	W =  90.000 deg,	P =   0.000 deg,	R =   90.000 deg
};
P[2220]{
   GP1:
	UF : 0, UT : 6,		CONFIG : 'N U T, 0, 0, 0',
	X =  162.027  mm,	Y =   -419.985  mm,	Z =   -309.000  mm,
	W =  90.000 deg,	P =   0.000 deg,	R =   90.000 deg
};
P[2221]{
   GP1:
	UF : 0, UT : 6,		CONFIG : 'N U T, 0, 0, 0',
	X =  163.134  mm,	Y =   -419.906  mm,	Z =   -309.000  mm,
	W =  90.000 deg,	P =   0.000 deg,	R =   90.000 deg
};
P[2222]{
   GP1:
	UF : 0, UT : 6,		CONFIG : 'N U T, 0, 0, 0',
	X =  164.129  mm,	Y =   -418.502  mm,	Z =   -309.000  mm,
	W =  90.000 deg,	P =   0.000 deg,	R =   90.000 deg
};
P[2223]{
   GP1:
	UF : 0, UT : 6,		CONFIG : 'N U T, 0, 0, 0',
	X =  165.168  mm,	Y =   -417.826  mm,	Z =   -309.000  mm,
	W =  90.000 deg,	P =   0.000 deg,	R =   90.000 deg
};
P[2224]{
   GP1:
	UF : 0, UT : 6,		CONFIG : 'N U T, 0, 0, 0',
	X =  166.318  mm,	Y =   -417.780  mm,	Z =   -309.000  mm,
	W =  90.000 deg,	P =   0.000 deg,	R =   90.000 deg
};
P[2225]{
   GP1:
	UF : 0, UT : 6,		CONFIG : 'N U T, 0, 0, 0',
	X =  166.758  mm,	Y =   -417.015  mm,	Z =   -319.532  mm,
	W =  90.000 deg,	P =   0.000 deg,	R =   90.000 deg
};
P[2226]{
   GP1:
	UF : 0, UT : 6,		CONFIG : 'N U T, 0, 0, 0',
	X =  167.771  mm,	Y =   -416.783  mm,	Z =   -309.000  mm,
	W =  90.000 deg,	P =   0.000 deg,	R =   90.000 deg
};
P[2227]{
   GP1:
	UF : 0, UT : 6,		CONFIG : 'N U T, 0, 0, 0',
	X =  170.041  mm,	Y =   -415.321  mm,	Z =   -309.050  mm,
	W =  90.000 deg,	P =   0.000 deg,	R =   90.000 deg
};
P[2228]{
   GP1:
	UF : 0, UT : 6,		CONFIG : 'N U T, 0, 0, 0',
	X =  171.103  mm,	Y =   -414.587  mm,	Z =   -309.100  mm,
	W =  90.000 deg,	P =   0.000 deg,	R =   90.000 deg
};
P[2229]{
   GP1:
	UF : 0, UT : 6,		CONFIG : 'N U T, 0, 0, 0',
	X =  172.428  mm,	Y =   -413.862  mm,	Z =   -309.000  mm,
	W =  90.000 deg,	P =   0.000 deg,	R =   90.000 deg
};
P[2230]{
   GP1:
	UF : 0, UT : 6,		CONFIG : 'N U T, 0, 0, 0',
	X =  173.442  mm,	Y =   -413.233  mm,	Z =   -309.000  mm,
	W =  90.000 deg,	P =   0.000 deg,	R =   90.000 deg
};
P[2231]{
   GP1:
	UF : 0, UT : 6,		CONFIG : 'N U T, 0, 0, 0',
	X =  174.583  mm,	Y =   -413.143  mm,	Z =   -309.000  mm,
	W =  90.000 deg,	P =   0.000 deg,	R =   90.000 deg
};
P[2232]{
   GP1:
	UF : 0, UT : 6,		CONFIG : 'N U T, 0, 0, 0',
	X =  175.789  mm,	Y =   -411.722  mm,	Z =   -309.100  mm,
	W =  90.000 deg,	P =   0.000 deg,	R =   90.000 deg
};
P[2233]{
   GP1:
	UF : 0, UT : 6,		CONFIG : 'N U T, 0, 0, 0',
	X =  177.245  mm,	Y =   -411.172  mm,	Z =   -309.100  mm,
	W =  90.000 deg,	P =   0.000 deg,	R =   90.000 deg
};
P[2234]{
   GP1:
	UF : 0, UT : 6,		CONFIG : 'N U T, 0, 0, 0',
	X =  178.353  mm,	Y =   -410.672  mm,	Z =   -309.000  mm,
	W =  90.000 deg,	P =   0.000 deg,	R =   90.000 deg
};
P[2235]{
   GP1:
	UF : 0, UT : 6,		CONFIG : 'N U T, 0, 0, 0',
	X =  179.204  mm,	Y =   -410.032  mm,	Z =   -309.000  mm,
	W =  90.000 deg,	P =   0.000 deg,	R =   90.000 deg
};
P[2236]{
   GP1:
	UF : 0, UT : 6,		CONFIG : 'N U T, 0, 0, 0',
	X =  180.330  mm,	Y =   -409.419  mm,	Z =   -309.000  mm,
	W =  90.000 deg,	P =   0.000 deg,	R =   90.000 deg
};
P[2237]{
   GP1:
	UF : 0, UT : 6,		CONFIG : 'N U T, 0, 0, 0',
	X =  181.471  mm,	Y =   -408.948  mm,	Z =   -309.100  mm,
	W =  90.000 deg,	P =   0.000 deg,	R =   90.000 deg
};
P[2238]{
   GP1:
	UF : 0, UT : 6,		CONFIG : 'N U T, 0, 0, 0',
	X =  181.883  mm,	Y =   -408.268  mm,	Z =   -309.000  mm,
	W =  90.000 deg,	P =   0.000 deg,	R =   90.000 deg
};
P[2239]{
   GP1:
	UF : 0, UT : 6,		CONFIG : 'N U T, 0, 0, 0',
	X =  182.859  mm,	Y =   -407.814  mm,	Z =   -309.100  mm,
	W =  90.000 deg,	P =   0.000 deg,	R =   90.000 deg
};
P[2240]{
   GP1:
	UF : 0, UT : 6,		CONFIG : 'N U T, 0, 0, 0',
	X =  183.947  mm,	Y =   -407.826  mm,	Z =   -309.000  mm,
	W =  90.000 deg,	P =   0.000 deg,	R =   90.000 deg
};
P[2241]{
   GP1:
	UF : 0, UT : 6,		CONFIG : 'N U T, 0, 0, 0',
	X =  184.634  mm,	Y =   -406.636  mm,	Z =   -309.000  mm,
	W =  90.000 deg,	P =   0.000 deg,	R =   90.000 deg
};
P[2242]{
   GP1:
	UF : 0, UT : 6,		CONFIG : 'N U T, 0, 0, 0',
	X =  185.431  mm,	Y =   -406.540  mm,	Z =   -309.000  mm,
	W =  90.000 deg,	P =   0.000 deg,	R =   90.000 deg
};
P[2243]{
   GP1:
	UF : 0, UT : 6,		CONFIG : 'N U T, 0, 0, 0',
	X =  186.214  mm,	Y =   -405.927  mm,	Z =   -309.000  mm,
	W =  90.000 deg,	P =   0.000 deg,	R =   90.000 deg
};
P[2244]{
   GP1:
	UF : 0, UT : 6,		CONFIG : 'N U T, 0, 0, 0',
	X =  187.090  mm,	Y =   -405.358  mm,	Z =   -309.100  mm,
	W =  90.000 deg,	P =   0.000 deg,	R =   90.000 deg
};
P[2245]{
   GP1:
	UF : 0, UT : 6,		CONFIG : 'N U T, 0, 0, 0',
	X =  188.145  mm,	Y =   -404.980  mm,	Z =   -309.100  mm,
	W =  90.000 deg,	P =   0.000 deg,	R =   90.000 deg
};
P[2246]{
   GP1:
	UF : 0, UT : 6,		CONFIG : 'N U T, 0, 0, 0',
	X =  189.942  mm,	Y =   -404.128  mm,	Z =   -320.766  mm,
	W =  90.000 deg,	P =   0.000 deg,	R =   90.000 deg
};
P[2247]{
   GP1:
	UF : 0, UT : 6,		CONFIG : 'N U T, 0, 0, 0',
	X =  190.660  mm,	Y =   -403.416  mm,	Z =   -309.100  mm,
	W =  90.000 deg,	P =   0.000 deg,	R =   90.000 deg
};
P[2248]{
   GP1:
	UF : 0, UT : 6,		CONFIG : 'N U T, 0, 0, 0',
	X =  191.337  mm,	Y =   -402.566  mm,	Z =   -309.000  mm,
	W =  90.000 deg,	P =   0.000 deg,	R =   90.000 deg
};
P[2249]{
   GP1:
	UF : 0, UT : 6,		CONFIG : 'N U T, 0, 0, 0',
	X =  192.932  mm,	Y =   -402.573  mm,	Z =   -309.100  mm,
	W =  90.000 deg,	P =   0.000 deg,	R =   90.000 deg
};
P[2250]{
   GP1:
	UF : 0, UT : 6,		CONFIG : 'N U T, 0, 0, 0',
	X =  193.978  mm,	Y =   -401.408  mm,	Z =   -309.000  mm,
	W =  90.000 deg,	P =   0.000 deg,	R =   90.000 deg
};
P[2251]{
   GP1:
	UF : 0, UT : 6,		CONFIG : 'N U T, 0, 0, 0',
	X =  195.193  mm,	Y =   -401.366  mm,	Z =   -309.000  mm,
	W =  90.000 deg,	P =   0.000 deg,	R =   90.000 deg
};
P[2252]{
   GP1:
	UF : 0, UT : 6,		CONFIG : 'N U T, 0, 0, 0',
	X =  196.007  mm,	Y =   -400.426  mm,	Z =   -309.000  mm,
	W =  90.000 deg,	P =   0.000 deg,	R =   90.000 deg
};
P[2253]{
   GP1:
	UF : 0, UT : 6,		CONFIG : 'N U T, 0, 0, 0',
	X =  196.731  mm,	Y =   -399.780  mm,	Z =   -309.000  mm,
	W =  90.000 deg,	P =   0.000 deg,	R =   90.000 deg
};
P[2254]{
   GP1:
	UF : 0, UT : 6,		CONFIG : 'N U T, 0, 0, 0',
	X =  198.078  mm,	Y =   -399.382  mm,	Z =   -309.000  mm,
	W =  90.000 deg,	P =   0.000 deg,	R =   90.000 deg
};
P[2255]{
   GP1:
	UF : 0, UT : 6,		CONFIG : 'N U T, 0, 0, 0',
	X =  198.385  mm,	Y =   -398.501  mm,	Z =   -326.028  mm,
	W =  90.000 deg,	P =   0.000 deg,	R =   90.000 deg
};
P[2256]{
   GP1:
	UF : 0, UT : 6,		CONFIG : 'N U T, 0, 0, 0',
	X =  200.033  mm,	Y =   -398.024  mm,	Z =   -316.284  mm,
	W =  90.000 deg,	P =   0.000 deg,	R =   90.000 deg
};
P[2257]{
   GP1:
	UF : 0, UT : 6,		CONFIG : 'N U T, 0, 0, 0',
	X =  200.824  mm,	Y =   -397.117  mm,	Z =   -309.000  mm,
	W =  90.000 deg,	P =   0.000 deg,	R =   90.000 deg
};
P[2258]{
   GP1:
	UF : 0, UT : 6,		CONFIG : 'N U T, 0, 0, 0',
	X =  201.991  mm,	Y =   -397.416  mm,	Z =   -309.965  mm,
	W =  90.000 deg,	P =   0.000 deg,	R =   90.000 deg
};
P[2259]{
   GP1:
	UF : 0, UT : 6,		CONFIG : 'N U T, 0, 0, 0',
	X =  202.754  mm,	Y =   -396.332  mm,	Z =   -309.000  mm,
	W =  90.000 deg,	P =   0.000 deg,	R =   90.000 deg
};
P[2260]{
   GP1:
	UF : 0, UT : 6,		CONFIG : 'N U T, 0, 0, 0',
	X =  204.058  mm,	Y =   -395.866  mm,	Z =   -309.000  mm,
	W =  90.000 deg,	P =   0.000 deg,	R =   90.000 deg
};
P[2261]{
   GP1:
	UF : 0, UT : 6,		CONFIG : 'N U T, 0, 0, 0',
	X =  204.928  mm,	Y =   -395.409  mm,	Z =   -309.000  mm,
	W =  90.000 deg,	P =   0.000 deg,	R =   90.000 deg
};
P[2262]{
   GP1:
	UF : 0, UT : 6,		CONFIG : 'N U T, 0, 0, 0',
	X =  205.473  mm,	Y =   -394.915  mm,	Z =   -309.000  mm,
	W =  90.000 deg,	P =   0.000 deg,	R =   90.000 deg
};
P[2263]{
   GP1:
	UF : 0, UT : 6,		CONFIG : 'N U T, 0, 0, 0',
	X =  206.213  mm,	Y =   -394.598  mm,	Z =   -309.000  mm,
	W =  90.000 deg,	P =   0.000 deg,	R =   90.000 deg
};
P[2264]{
   GP1:
	UF : 0, UT : 6,		CONFIG : 'N U T, 0, 0, 0',
	X =  207.135  mm,	Y =   -393.818  mm,	Z =   -309.000  mm,
	W =  90.000 deg,	P =   0.000 deg,	R =   90.000 deg
};
P[2265]{
   GP1:
	UF : 0, UT : 6,		CONFIG : 'N U T, 0, 0, 0',
	X =  208.850  mm,	Y =   -393.016  mm,	Z =   -309.000  mm,
	W =  90.000 deg,	P =   0.000 deg,	R =   90.000 deg
};
P[2266]{
   GP1:
	UF : 0, UT : 6,		CONFIG : 'N U T, 0, 0, 0',
	X =  210.631  mm,	Y =   -392.153  mm,	Z =   -309.000  mm,
	W =  90.000 deg,	P =   0.000 deg,	R =   90.000 deg
};
P[2267]{
   GP1:
	UF : 0, UT : 6,		CONFIG : 'N U T, 0, 0, 0',
	X =  211.388  mm,	Y =   -391.923  mm,	Z =   -309.000  mm,
	W =  90.000 deg,	P =   0.000 deg,	R =   90.000 deg
};
P[2268]{
   GP1:
	UF : 0, UT : 6,		CONFIG : 'N U T, 0, 0, 0',
	X =  211.934  mm,	Y =   -391.289  mm,	Z =   -309.000  mm,
	W =  90.000 deg,	P =   0.000 deg,	R =   90.000 deg
};
P[2269]{
   GP1:
	UF : 0, UT : 6,		CONFIG : 'N U T, 0, 0, 0',
	X =  213.387  mm,	Y =   -390.357  mm,	Z =   -309.000  mm,
	W =  90.000 deg,	P =   0.000 deg,	R =   90.000 deg
};
P[2270]{
   GP1:
	UF : 0, UT : 6,		CONFIG : 'N U T, 0, 0, 0',
	X =  214.208  mm,	Y =   -389.492  mm,	Z =   -309.100  mm,
	W =  90.000 deg,	P =   0.000 deg,	R =   90.000 deg
};
P[2271]{
   GP1:
	UF : 0, UT : 6,		CONFIG : 'N U T, 0, 0, 0',
	X =  215.354  mm,	Y =   -389.141  mm,	Z =   -309.000  mm,
	W =  90.000 deg,	P =   0.000 deg,	R =   90.000 deg
};
P[2272]{
   GP1:
	UF : 0, UT : 6,		CONFIG : 'N U T, 0, 0, 0',
	X =  216.178  mm,	Y =   -388.626  mm,	Z =   -309.000  mm,
	W =  90.000 deg,	P =   0.000 deg,	R =   90.000 deg
};
P[2273]{
   GP1:
	UF : 0, UT : 6,		CONFIG : 'N U T, 0, 0, 0',
	X =  217.380  mm,	Y =   -387.993  mm,	Z =   -309.100  mm,
	W =  90.000 deg,	P =   0.000 deg,	R =   90.000 deg
};
P[2274]{
   GP1:
	UF : 0, UT : 6,		CONFIG : 'N U T, 0, 0, 0',
	X =  218.562  mm,	Y =   -387.083  mm,	Z =   -309.000  mm,
	W =  90.000 deg,	P =   0.000 deg,	R =   90.000 deg
};
P[2275]{
   GP1:
	UF : 0, UT : 6,		CONFIG : 'N U T, 0, 0, 0',
	X =  219.941  mm,	Y =   -386.539  mm,	Z =   -309.100  mm,
	W =  90.000 deg,	P =   0.000 deg,	R =   90.000 deg
};
P[2276]{
   GP1:
	UF : 0, UT : 6,		CONFIG : 'N U T, 0, 0, 0',
	X =  221.209  mm,	Y =   -386.213  mm,	Z =   -309.000  mm,
	W =  90.000 deg,	P =   0.000 deg,	R =   90.000 deg
};
P[2277]{
   GP1:
	UF : 0, UT : 6,		CONFIG : 'N U T, 0, 0, 0',
	X =  222.109  mm,	Y =   -385.589  mm,	Z =   -309.100  mm,
	W =  90.000 deg,	P =   0.000 deg,	R =   90.000 deg
};
P[2278]{
   GP1:
	UF : 0, UT : 6,		CONFIG : 'N U T, 0, 0, 0',
	X =  222.648  mm,	Y =   -384.774  mm,	Z =   -309.000  mm,
	W =  90.000 deg,	P =   0.000 deg,	R =   90.000 deg
};
P[2279]{
   GP1:
	UF : 0, UT : 6,		CONFIG : 'N U T, 0, 0, 0',
	X =  223.873  mm,	Y =   -384.552  mm,	Z =   -309.100  mm,
	W =  90.000 deg,	P =   0.000 deg,	R =   90.000 deg
};
P[2280]{
   GP1:
	UF : 0, UT : 6,		CONFIG : 'N U T, 0, 0, 0',
	X =  224.699  mm,	Y =   -384.405  mm,	Z =   -309.000  mm,
	W =  90.000 deg,	P =   0.000 deg,	R =   90.000 deg
};
P[2281]{
   GP1:
	UF : 0, UT : 6,		CONFIG : 'N U T, 0, 0, 0',
	X =  225.007  mm,	Y =   -383.425  mm,	Z =   -309.000  mm,
	W =  90.000 deg,	P =   0.000 deg,	R =   90.000 deg
};
P[2282]{
   GP1:
	UF : 0, UT : 6,		CONFIG : 'N U T, 0, 0, 0',
	X =  225.789  mm,	Y =   -383.130  mm,	Z =   -309.100  mm,
	W =  90.000 deg,	P =   0.000 deg,	R =   90.000 deg
};
P[2283]{
   GP1:
	UF : 0, UT : 6,		CONFIG : 'N U T, 0, 0, 0',
	X =  227.034  mm,	Y =   -382.387  mm,	Z =   -309.000  mm,
	W =  90.000 deg,	P =   0.000 deg,	R =   90.000 deg
};
P[2284]{
   GP1:
	UF : 0, UT : 6,		CONFIG : 'N U T, 0, 0, 0',
	X =  228.283  mm,	Y =   -382.023  mm,	Z =   -309.100  mm,
	W =  90.000 deg,	P =   0.000 deg,	R =   90.000 deg
};
P[2285]{
   GP1:
	UF : 0, UT : 6,		CONFIG : 'N U T, 0, 0, 0',
	X =  228.695  mm,	Y =   -381.182  mm,	Z =   -309.000  mm,
	W =  90.000 deg,	P =   0.000 deg,	R =   90.000 deg
};
P[2286]{
   GP1:
	UF : 0, UT : 6,		CONFIG : 'N U T, 0, 0, 0',
	X =  229.542  mm,	Y =   -381.395  mm,	Z =   -317.391  mm,
	W =  90.000 deg,	P =   0.000 deg,	R =   90.000 deg
};
P[2287]{
   GP1:
	UF : 0, UT : 6,		CONFIG : 'N U T, 0, 0, 0',
	X =  230.093  mm,	Y =   -380.521  mm,	Z =   -309.000  mm,
	W =  90.000 deg,	P =   0.000 deg,	R =   90.000 deg
};
P[2288]{
   GP1:
	UF : 0, UT : 6,		CONFIG : 'N U T, 0, 0, 0',
	X =  231.166  mm,	Y =   -380.525  mm,	Z =   -309.000  mm,
	W =  90.000 deg,	P =   0.000 deg,	R =   90.000 deg
};
P[2289]{
   GP1:
	UF : 0, UT : 6,		CONFIG : 'N U T, 0, 0, 0',
	X =  232.025  mm,	Y =   -380.117  mm,	Z =   -309.100  mm,
	W =  90.000 deg,	P =   0.000 deg,	R =   90.000 deg
};
P[2290]{
   GP1:
	UF : 0, UT : 6,		CONFIG : 'N U T, 0, 0, 0',
	X =  232.780  mm,	Y =   -378.922  mm,	Z =   -312.031  mm,
	W =  90.000 deg,	P =   0.000 deg,	R =   90.000 deg
};
P[2291]{
   GP1:
	UF : 0, UT : 6,		CONFIG : 'N U T, 0, 0, 0',
	X =  233.938  mm,	Y =   -378.455  mm,	Z =   -309.100  mm,
	W =  90.000 deg,	P =   0.000 deg,	R =   90.000 deg
};
P[2292]{
   GP1:
	UF : 0, UT : 6,		CONFIG : 'N U T, 0, 0, 0',
	X =  234.858  mm,	Y =   -378.108  mm,	Z =   -309.100  mm,
	W =  90.000 deg,	P =   0.000 deg,	R =   90.000 deg
};
P[2293]{
   GP1:
	UF : 0, UT : 6,		CONFIG : 'N U T, 0, 0, 0',
	X =  236.276  mm,	Y =   -377.628  mm,	Z =   -309.100  mm,
	W =  90.000 deg,	P =   0.000 deg,	R =   90.000 deg
};
P[2294]{
   GP1:
	UF : 0, UT : 6,		CONFIG : 'N U T, 0, 0, 0',
	X =  236.587  mm,	Y =   -376.933  mm,	Z =   -309.100  mm,
	W =  90.000 deg,	P =   0.000 deg,	R =   90.000 deg
};
P[2295]{
   GP1:
	UF : 0, UT : 6,		CONFIG : 'N U T, 0, 0, 0',
	X =  238.157  mm,	Y =   -375.744  mm,	Z =   -309.358  mm,
	W =  90.000 deg,	P =   0.000 deg,	R =   90.000 deg
};
P[2296]{
   GP1:
	UF : 0, UT : 6,		CONFIG : 'N U T, 0, 0, 0',
	X =  239.179  mm,	Y =   -375.642  mm,	Z =   -309.000  mm,
	W =  90.000 deg,	P =   0.000 deg,	R =   90.000 deg
};
P[2297]{
   GP1:
	UF : 0, UT : 6,		CONFIG : 'N U T, 0, 0, 0',
	X =  239.950  mm,	Y =   -375.070  mm,	Z =   -309.000  mm,
	W =  90.000 deg,	P =   0.000 deg,	R =   90.000 deg
};
P[2298]{
   GP1:
	UF : 0, UT : 6,		CONFIG : 'N U T, 0, 0, 0',
	X =  241.158  mm,	Y =   -374.648  mm,	Z =   -309.000  mm,
	W =  90.000 deg,	P =   0.000 deg,	R =   90.000 deg
};
P[2299]{
   GP1:
	UF : 0, UT : 6,		CONFIG : 'N U T, 0, 0, 0',
	X =  241.532  mm,	Y =   -373.876  mm,	Z =   -309.000  mm,
	W =  90.000 deg,	P =   0.000 deg,	R =   90.000 deg
};
P[2300]{
   GP1:
	UF : 0, UT : 6,		CONFIG : 'N U T, 0, 0, 0',
	X =  242.528  mm,	Y =   -373.702  mm,	Z =   -309.000  mm,
	W =  90.000 deg,	P =   0.000 deg,	R =   90.000 deg
};
P[2301]{
   GP1:
	UF : 0, UT : 6,		CONFIG : 'N U T, 0, 0, 0',
	X =  243.372  mm,	Y =   -373.133  mm,	Z =   -309.000  mm,
	W =  90.000 deg,	P =   0.000 deg,	R =   90.000 deg
};
P[2302]{
   GP1:
	UF : 0, UT : 6,		CONFIG : 'N U T, 0, 0, 0',
	X =  244.205  mm,	Y =   -372.323  mm,	Z =   -309.000  mm,
	W =  90.000 deg,	P =   0.000 deg,	R =   90.000 deg
};
P[2303]{
   GP1:
	UF : 0, UT : 6,		CONFIG : 'N U T, 0, 0, 0',
	X =  245.156  mm,	Y =   -371.907  mm,	Z =   -309.000  mm,
	W =  90.000 deg,	P =   0.000 deg,	R =   90.000 deg
};
P[2304]{
   GP1:
	UF : 0, UT : 6,		CONFIG : 'N U T, 0, 0, 0',
	X =  245.843  mm,	Y =   -371.625  mm,	Z =   -309.000  mm,
	W =  90.000 deg,	P =   0.000 deg,	R =   90.000 deg
};
P[2305]{
   GP1:
	UF : 0, UT : 6,		CONFIG : 'N U T, 0, 0, 0',
	X =  246.532  mm,	Y =   -371.024  mm,	Z =   -309.000  mm,
	W =  90.000 deg,	P =   0.000 deg,	R =   90.000 deg
};
P[2306]{
   GP1:
	UF : 0, UT : 6,		CONFIG : 'N U T, 0, 0, 0',
	X =  247.811  mm,	Y =   -370.550  mm,	Z =   -309.100  mm,
	W =  90.000 deg,	P =   0.000 deg,	R =   90.000 deg
};
P[2307]{
   GP1:
	UF : 0, UT : 6,		CONFIG : 'N U T, 0, 0, 0',
	X =  248.776  mm,	Y =   -369.508  mm,	Z =   -309.000  mm,
	W =  90.000 deg,	P =   0.000 deg,	R =   90.000 deg
};
P[2308]{
   GP1:
	UF : 0, UT : 6,		CONFIG : 'N U T, 0, 0, 0',
	X =  249.514  mm,	Y =   -369.514  mm,	Z =   -309.000  mm,
	W =  90.000 deg,	P =   0.000 deg,	R =   90.000 deg
};
P[2309]{
   GP1:
	UF : 0, UT : 6,		CONFIG : 'N U T, 0, 0, 0',
	X =  250.806  mm,	Y =   -368.738  mm,	Z =   -309.000  mm,
	W =  90.000 deg,	P =   0.000 deg,	R =   90.000 deg
};
P[2310]{
   GP1:
	UF : 0, UT : 6,		CONFIG : 'N U T, 0, 0, 0',
	X =  252.019  mm,	Y =   -367.771  mm,	Z =   -309.100  mm,
	W =  90.000 deg,	P =   0.000 deg,	R =   90.000 deg
};
P[2311]{
   GP1:
	UF : 0, UT : 6,		CONFIG : 'N U T, 0, 0, 0',
	X =  252.899  mm,	Y =   -367.564  mm,	Z =   -309.000  mm,
	W =  90.000 deg,	P =   0.000 deg,	R =   90.000 deg
};
P[2312]{
   GP1:
	UF : 0, UT : 6,		CONFIG : 'N U T, 0, 0, 0',
	X =  253.595  mm,	Y =   -366.661  mm,	Z =   -309.100  mm,
	W =  90.000 deg,	P =   0.000 deg,	R =   90.000 deg
};
P[2313]{
   GP1:
	UF : 0, UT : 6,		CONFIG : 'N U T, 0, 0, 0',
	X =  254.507  mm,	Y =   -366.511  mm,	Z =   -309.100  mm,
	W =  90.000 deg,	P =   0.000 deg,	R =   90.000 deg
};
P[2314]{
   GP1:
	UF : 0, UT : 6,		CONFIG : 'N U T, 0, 0, 0',
	X =  255.333  mm,	Y =   -366.262  mm,	Z =   -309.100  mm,
	W =  90.000 deg,	P =   0.000 deg,	R =   90.000 deg
};
P[2315]{
   GP1:
	UF : 0, UT : 6,		CONFIG : 'N U T, 0, 0, 0',
	X =  256.090  mm,	Y =   -365.548  mm,	Z =   -309.000  mm,
	W =  90.000 deg,	P =   0.000 deg,	R =   90.000 deg
};
P[2316]{
   GP1:
	UF : 0, UT : 6,		CONFIG : 'N U T, 0, 0, 0',
	X =  257.424  mm,	Y =   -365.316  mm,	Z =   -309.100  mm,
	W =  90.000 deg,	P =   0.000 deg,	R =   90.000 deg
};
P[2317]{
   GP1:
	UF : 0, UT : 6,		CONFIG : 'N U T, 0, 0, 0',
	X =  258.438  mm,	Y =   -364.741  mm,	Z =   -309.000  mm,
	W =  90.000 deg,	P =   0.000 deg,	R =   90.000 deg
};
P[2318]{
   GP1:
	UF : 0, UT : 6,		CONFIG : 'N U T, 0, 0, 0',
	X =  259.191  mm,	Y =   -364.046  mm,	Z =   -309.000  mm,
	W =  90.000 deg,	P =   0.000 deg,	R =   90.000 deg
};
P[2319]{
   GP1:
	UF : 0, UT : 6,		CONFIG : 'N U T, 0, 0, 0',
	X =  259.933  mm,	Y =   -363.698  mm,	Z =   -309.000  mm,
	W =  90.000 deg,	P =   0.000 deg,	R =   90.000 deg
};
P[2320]{
   GP1:
	UF : 0, UT : 6,		CONFIG : 'N U T, 0, 0, 0',
	X =  260.785  mm,	Y =   -362.823  mm,	Z =   -309.100  mm,
	W =  90.000 deg,	P =   0.000 deg,	R =   90.000 deg
};
P[2321]{
   GP1:
	UF : 0, UT : 6,		CONFIG : 'N U T, 0, 0, 0',
	X =  261.653  mm,	Y =   -362.588  mm,	Z =   -309.100  mm,
	W =  90.000 deg,	P =   0.000 deg,	R =   90.000 deg
};
P[2322]{
   GP1:
	UF : 0, UT : 6,		CONFIG : 'N U T, 0, 0, 0',
	X =  262.366  mm,	Y =   -362.246  mm,	Z =   -309.100  mm,
	W =  90.000 deg,	P =   0.000 deg,	R =   90.000 deg
};
P[2323]{
   GP1:
	UF : 0, UT : 6,		CONFIG : 'N U T, 0, 0, 0',
	X =  262.884  mm,	Y =   -361.294  mm,	Z =   -316.202  mm,
	W =  90.000 deg,	P =   0.000 deg,	R =   90.000 deg
};
P[2324]{
   GP1:
	UF : 0, UT : 6,		CONFIG : 'N U T, 0, 0, 0',
	X =  263.871  mm,	Y =   -361.061  mm,	Z =   -309.000  mm,
	W =  90.000 deg,	P =   0.000 deg,	R =   90.000 deg
};
P[2325]{
   GP1:
	UF : 0, UT : 6,		CONFIG : 'N U T, 0, 0, 0',
	X =  265.337  mm,	Y =   -360.018  mm,	Z =   -309.000  mm,
	W =  90.000 deg,	P =   0.000 deg,	R =   90.000 deg
};
P[2326]{
   GP1:
	UF : 0, UT : 6,		CONFIG : 'N U T, 0, 0, 0',
	X =  266.134  mm,	Y =   -360.454  mm,	Z =   -309.000  mm,
	W =  90.000 deg,	P =   0.000 deg,	R =   90.000 deg
};
P[2327]{
   GP1:
	UF : 0, UT : 6,		CONFIG : 'N U T, 0, 0, 0',
	X =  266.637  mm,	Y =   -359.522  mm,	Z =   -309.000  mm,
	W =  90.000 deg,	P =   0.000 deg,	R =   90.000 deg
};
P[2328]{
   GP1:
	UF : 0, UT : 6,		CONFIG : 'N U T, 0, 0, 0',
	X =  267.740  mm,	Y =   -359.082  mm,	Z =   -309.000  mm,
	W =  90.000 deg,	P =   0.000 deg,	R =   90.000 deg
};
P[2329]{
   GP1:
	UF : 0, UT : 6,		CONFIG : 'N U T, 0, 0, 0',
	X =  268.555  mm,	Y =   -358.336  mm,	Z =   -309.000  mm,
	W =  90.000 deg,	P =   0.000 deg,	R =   90.000 deg
};
P[2330]{
   GP1:
	UF : 0, UT : 6,		CONFIG : 'N U T, 0, 0, 0',
	X =  269.329  mm,	Y =   -357.992  mm,	Z =   -309.100  mm,
	W =  90.000 deg,	P =   0.000 deg,	R =   90.000 deg
};
P[2331]{
   GP1:
	UF : 0, UT : 6,		CONFIG : 'N U T, 0, 0, 0',
	X =  270.292  mm,	Y =   -357.362  mm,	Z =   -309.100  mm,
	W =  90.000 deg,	P =   0.000 deg,	R =   90.000 deg
};
P[2332]{
   GP1:
	UF : 0, UT : 6,		CONFIG : 'N U T, 0, 0, 0',
	X =  271.290  mm,	Y =   -357.019  mm,	Z =   -309.100  mm,
	W =  90.000 deg,	P =   0.000 deg,	R =   90.000 deg
};
P[2333]{
   GP1:
	UF : 0, UT : 6,		CONFIG : 'N U T, 0, 0, 0',
	X =  272.007  mm,	Y =   -356.490  mm,	Z =   -309.000  mm,
	W =  90.000 deg,	P =   0.000 deg,	R =   90.000 deg
};
P[2334]{
   GP1:
	UF : 0, UT : 6,		CONFIG : 'N U T, 0, 0, 0',
	X =  273.145  mm,	Y =   -356.367  mm,	Z =   -309.000  mm,
	W =  90.000 deg,	P =   0.000 deg,	R =   90.000 deg
};
P[2335]{
   GP1:
	UF : 0, UT : 6,		CONFIG : 'N U T, 0, 0, 0',
	X =  273.848  mm,	Y =   -355.937  mm,	Z =   -309.000  mm,
	W =  90.000 deg,	P =   0.000 deg,	R =   90.000 deg
};
P[2336]{
   GP1:
	UF : 0, UT : 6,		CONFIG : 'N U T, 0, 0, 0',
	X =  274.960  mm,	Y =   -354.619  mm,	Z =   -309.100  mm,
	W =  90.000 deg,	P =   0.000 deg,	R =   90.000 deg
};
P[2337]{
   GP1:
	UF : 0, UT : 6,		CONFIG : 'N U T, 0, 0, 0',
	X =  275.596  mm,	Y =   -354.271  mm,	Z =   -309.000  mm,
	W =  90.000 deg,	P =   0.000 deg,	R =   90.000 deg
};
P[2338]{
   GP1:
	UF : 0, UT : 6,		CONFIG : 'N U T, 0, 0, 0',
	X =  277.136  mm,	Y =   -353.257  mm,	Z =   -309.100  mm,
	W =  90.000 deg,	P =   0.000 deg,	R =   90.000 deg
};
P[2339]{
   GP1:
	UF : 0, UT : 6,		CONFIG : 'N U T, 0, 0, 0',
	X =  278.520  mm,	Y =   -353.282  mm,	Z =   -309.000  mm,
	W =  90.000 deg,	P =   0.000 deg,	R =   90.000 deg
};
P[2340]{
   GP1:
	UF : 0, UT : 6,		CONFIG : 'N U T, 0, 0, 0',
	X =  278.928  mm,	Y =   -352.576  mm,	Z =   -309.000  mm,
	W =  90.000 deg,	P =   0.000 deg,	R =   90.000 deg
};
P[2341]{
   GP1:
	UF : 0, UT : 6,		CONFIG : 'N U T, 0, 0, 0',
	X =  279.617  mm,	Y =   -352.027  mm,	Z =   -309.100  mm,
	W =  90.000 deg,	P =   0.000 deg,	R =   90.000 deg
};
P[2342]{
   GP1:
	UF : 0, UT : 6,		CONFIG : 'N U T, 0, 0, 0',
	X =  280.471  mm,	Y =   -351.553  mm,	Z =   -309.000  mm,
	W =  90.000 deg,	P =   0.000 deg,	R =   90.000 deg
};
P[2343]{
   GP1:
	UF : 0, UT : 6,		CONFIG : 'N U T, 0, 0, 0',
	X =  281.634  mm,	Y =   -351.238  mm,	Z =   -311.253  mm,
	W =  90.000 deg,	P =   0.000 deg,	R =   90.000 deg
};
P[2344]{
   GP1:
	UF : 0, UT : 6,		CONFIG : 'N U T, 0, 0, 0',
	X =  282.316  mm,	Y =   -350.305  mm,	Z =   -309.100  mm,
	W =  90.000 deg,	P =   0.000 deg,	R =   90.000 deg
};
P[2345]{
   GP1:
	UF : 0, UT : 6,		CONFIG : 'N U T, 0, 0, 0',
	X =  283.514  mm,	Y =   -349.893  mm,	Z =   -309.000  mm,
	W =  90.000 deg,	P =   0.000 deg,	R =   90.000 deg
};
P[2346]{
   GP1:
	UF : 0, UT : 6,		CONFIG : 'N U T, 0, 0, 0',
	X =  284.175  mm,	Y =   -349.618  mm,	Z =   -309.000  mm,
	W =  90.000 deg,	P =   0.000 deg,	R =   90.000 deg
};
P[2347]{
   GP1:
	UF : 0, UT : 6,		CONFIG : 'N U T, 0, 0, 0',
	X =  285.213  mm,	Y =   -348.612  mm,	Z =   -309.000  mm,
	W =  90.000 deg,	P =   0.000 deg,	R =   90.000 deg
};
P[2348]{
   GP1:
	UF : 0, UT : 6,		CONFIG : 'N U T, 0, 0, 0',
	X =  285.963  mm,	Y =   -348.399  mm,	Z =   -309.000  mm,
	W =  90.000 deg,	P =   0.000 deg,	R =   90.000 deg
};
P[2349]{
   GP1:
	UF : 0, UT : 6,		CONFIG : 'N U T, 0, 0, 0',
	X =  287.314  mm,	Y =   -348.159  mm,	Z =   -309.000  mm,
	W =  90.000 deg,	P =   0.000 deg,	R =   90.000 deg
};
P[2350]{
   GP1:
	UF : 0, UT : 6,		CONFIG : 'N U T, 0, 0, 0',
	X =  287.337  mm,	Y =   -347.240  mm,	Z =   -309.100  mm,
	W =  90.000 deg,	P =   0.000 deg,	R =   90.000 deg
};
P[2351]{
   GP1:
	UF : 0, UT : 6,		CONFIG : 'N U T, 0, 0, 0',
	X =  288.627  mm,	Y =   -346.986  mm,	Z =   -309.000  mm,
	W =  90.000 deg,	P =   0.000 deg,	R =   90.000 deg
};
P[2352]{
   GP1:
	UF : 0, UT : 6,		CONFIG : 'N U T, 0, 0, 0',
	X =  289.364  mm,	Y =   -346.288  mm,	Z =   -309.000  mm,
	W =  90.000 deg,	P =   0.000 deg,	R =   90.000 deg
};
P[2353]{
   GP1:
	UF : 0, UT : 6,		CONFIG : 'N U T, 0, 0, 0',
	X =  290.316  mm,	Y =   -346.193  mm,	Z =   -309.000  mm,
	W =  90.000 deg,	P =   0.000 deg,	R =   90.000 deg
};
P[2354]{
   GP1:
	UF : 0, UT : 6,		CONFIG : 'N U T, 0, 0, 0',
	X =  291.002  mm,	Y =   -345.750  mm,	Z =   -309.100  mm,
	W =  90.000 deg,	P =   0.000 deg,	R =   90.000 deg
};
P[2355]{
   GP1:
	UF : 0, UT : 6,		CONFIG : 'N U T, 0, 0, 0',
	X =  291.794  mm,	Y =   -344.911  mm,	Z =   -309.000  mm,
	W =  90.000 deg,	P =   0.000 deg,	R =   90.000 deg
};
P[2356]{
   GP1:
	UF : 0, UT : 6,		CONFIG : 'N U T, 0, 0, 0',
	X =  292.956  mm,	Y =   -344.206  mm,	Z =   -309.000  mm,
	W =  90.000 deg,	P =   0.000 deg,	R =   90.000 deg
};
P[2357]{
   GP1:
	UF : 0, UT : 6,		CONFIG : 'N U T, 0, 0, 0',
	X =  293.754  mm,	Y =   -344.018  mm,	Z =   -309.000  mm,
	W =  90.000 deg,	P =   0.000 deg,	R =   90.000 deg
};
P[2358]{
   GP1:
	UF : 0, UT : 6,		CONFIG : 'N U T, 0, 0, 0',
	X =  294.737  mm,	Y =   -343.356  mm,	Z =   -309.000  mm,
	W =  90.000 deg,	P =   0.000 deg,	R =   90.000 deg
};
P[2359]{
   GP1:
	UF : 0, UT : 6,		CONFIG : 'N U T, 0, 0, 0',
	X =  295.484  mm,	Y =   -343.409  mm,	Z =   -309.100  mm,
	W =  90.000 deg,	P =   0.000 deg,	R =   90.000 deg
};
P[2360]{
   GP1:
	UF : 0, UT : 6,		CONFIG : 'N U T, 0, 0, 0',
	X =  296.361  mm,	Y =   -342.329  mm,	Z =   -309.100  mm,
	W =  90.000 deg,	P =   0.000 deg,	R =   90.000 deg
};
P[2361]{
   GP1:
	UF : 0, UT : 6,		CONFIG : 'N U T, 0, 0, 0',
	X =  297.270  mm,	Y =   -342.106  mm,	Z =   -309.000  mm,
	W =  90.000 deg,	P =   0.000 deg,	R =   90.000 deg
};
P[2362]{
   GP1:
	UF : 0, UT : 6,		CONFIG : 'N U T, 0, 0, 0',
	X =  297.979  mm,	Y =   -341.489  mm,	Z =   -309.000  mm,
	W =  90.000 deg,	P =   0.000 deg,	R =   90.000 deg
};
P[2363]{
   GP1:
	UF : 0, UT : 6,		CONFIG : 'N U T, 0, 0, 0',
	X =  299.030  mm,	Y =   -341.273  mm,	Z =   -309.000  mm,
	W =  90.000 deg,	P =   0.000 deg,	R =   90.000 deg
};
P[2364]{
   GP1:
	UF : 0, UT : 6,		CONFIG : 'N U T, 0, 0, 0',
	X =  299.696  mm,	Y =   -340.673  mm,	Z =   -309.000  mm,
	W =  90.000 deg,	P =   0.000 deg,	R =   90.000 deg
};
P[2365]{
   GP1:
	UF : 0, UT : 6,		CONFIG : 'N U T, 0, 0, 0',
	X =  300.718  mm,	Y =   -340.119  mm,	Z =   -319.803  mm,
	W =  90.000 deg,	P =   0.000 deg,	R =   90.000 deg
};
P[2366]{
   GP1:
	UF : 0, UT : 6,		CONFIG : 'N U T, 0, 0, 0',
	X =  301.894  mm,	Y =   -339.747  mm,	Z =   -309.100  mm,
	W =  90.000 deg,	P =   0.000 deg,	R =   90.000 deg
};
P[2367]{
   GP1:
	UF : 0, UT : 6,		CONFIG : 'N U T, 0, 0, 0',
	X =  302.729  mm,	Y =   -338.906  mm,	Z =   -309.000  mm,
	W =  90.000 deg,	P =   0.000 deg,	R =   90.000 deg
};
P[2368]{
   GP1:
	UF : 0, UT : 6,		CONFIG : 'N U T, 0, 0, 0',
	X =  303.804  mm,	Y =   -338.088  mm,	Z =   -309.000  mm,
	W =  90.000 deg,	P =   0.000 deg,	R =   90.000 deg
};
P[2369]{
   GP1:
	UF : 0, UT : 6,		CONFIG : 'N U T, 0, 0, 0',
	X =  310.971  mm,	Y =   -351.819  mm,	Z =   -309.000  mm,
	W =  90.000 deg,	P =   0.000 deg,	R =   90.000 deg
};
P[2370]{
   GP1:
	UF : 0, UT : 6,		CONFIG : 'N U T, 0, 0, 0',
	X =  309.813  mm,	Y =   -351.976  mm,	Z =   -309.000  mm,
	W =  90.000 deg,	P =   0.000 deg,	R =   90.000 deg
};
P[2371]{
   GP1:
	UF : 0, UT : 6,		CONFIG : 'N U T, 0, 0, 0',
	X =  308.722  mm,	Y =   -352.211  mm,	Z =   -309.100  mm,
	W =  90.000 deg,	P =   0.000 deg,	R =   90.000 deg
};
P[2372]{
   GP1:
	UF : 0, UT : 6,		CONFIG : 'N U T, 0, 0, 0',
	X =  308.350  mm,	Y =   -353.070  mm,	Z =   -309.100  mm,
	W =  90.000 deg,	P =   0.000 deg,	R =   90.000 deg
};
P[2373]{
   GP1:
	UF : 0, UT : 6,		CONFIG : 'N U T, 0, 0, 0',
	X =  307.532  mm,	Y =   -353.357  mm,	Z =   -309.000  mm,
	W =  90.000 deg,	P =   0.000 deg,	R =   90.000 deg
};
P[2374]{
   GP1:
	UF : 0, UT : 6,		CONFIG : 'N U T, 0, 0, 0',
	X =  306.695  mm,	Y =   -353.779  mm,	Z =   -309.000  mm,
	W =  90.000 deg,	P =   0.000 deg,	R =   90.000 deg
};
P[2375]{
   GP1:
	UF : 0, UT : 6,		CONFIG : 'N U T, 0, 0, 0',
	X =  305.389  mm,	Y =   -354.596  mm,	Z =   -309.100  mm,
	W =  90.000 deg,	P =   0.000 deg,	R =   90.000 deg
};
P[2376]{
   GP1:
	UF : 0, UT : 6,		CONFIG : 'N U T, 0, 0, 0',
	X =  304.981  mm,	Y =   -355.075  mm,	Z =   -309.000  mm,
	W =  90.000 deg,	P =   0.000 deg,	R =   90.000 deg
};
P[2377]{
   GP1:
	UF : 0, UT : 6,		CONFIG : 'N U T, 0, 0, 0',
	X =  303.978  mm,	Y =   -355.166  mm,	Z =   -309.000  mm,
	W =  90.000 deg,	P =   0.000 deg,	R =   90.000 deg
};
P[2378]{
   GP1:
	UF : 0, UT : 6,		CONFIG : 'N U T, 0, 0, 0',
	X =  301.677  mm,	Y =   -356.495  mm,	Z =   -309.000  mm,
	W =  90.000 deg,	P =   0.000 deg,	R =   90.000 deg
};
P[2379]{
   GP1:
	UF : 0, UT : 6,		CONFIG : 'N U T, 0, 0, 0',
	X =  300.845  mm,	Y =   -357.283  mm,	Z =   -309.100  mm,
	W =  90.000 deg,	P =   0.000 deg,	R =   90.000 deg
};
P[2380]{
   GP1:
	UF : 0, UT : 6,		CONFIG : 'N U T, 0, 0, 0',
	X =  300.093  mm,	Y =   -357.409  mm,	Z =   -309.000  mm,
	W =  90.000 deg,	P =   0.000 deg,	R =   90.000 deg
};
P[2381]{
   GP1:
	UF : 0, UT : 6,		CONFIG : 'N U T, 0, 0, 0',
	X =  299.538  mm,	Y =   -358.401  mm,	Z =   -309.100  mm,
	W =  90.000 deg,	P =   0.000 deg,	R =   90.000 deg
};
P[2382]{
   GP1:
	UF : 0, UT : 6,		CONFIG : 'N U T, 0, 0, 0',
	X =  298.465  mm,	Y =   -358.133  mm,	Z =   -309.100  mm,
	W =  90.000 deg,	P =   0.000 deg,	R =   90.000 deg
};
P[2383]{
   GP1:
	UF : 0, UT : 6,		CONFIG : 'N U T, 0, 0, 0',
	X =  298.085  mm,	Y =   -359.062  mm,	Z =   -309.000  mm,
	W =  90.000 deg,	P =   0.000 deg,	R =   90.000 deg
};
P[2384]{
   GP1:
	UF : 0, UT : 6,		CONFIG : 'N U T, 0, 0, 0',
	X =  296.597  mm,	Y =   -359.957  mm,	Z =   -318.233  mm,
	W =  90.000 deg,	P =   0.000 deg,	R =   90.000 deg
};
P[2385]{
   GP1:
	UF : 0, UT : 6,		CONFIG : 'N U T, 0, 0, 0',
	X =  295.833  mm,	Y =   -359.739  mm,	Z =   -309.100  mm,
	W =  90.000 deg,	P =   0.000 deg,	R =   90.000 deg
};
P[2386]{
   GP1:
	UF : 0, UT : 6,		CONFIG : 'N U T, 0, 0, 0',
	X =  295.353  mm,	Y =   -360.605  mm,	Z =   -309.000  mm,
	W =  90.000 deg,	P =   0.000 deg,	R =   90.000 deg
};
P[2387]{
   GP1:
	UF : 0, UT : 6,		CONFIG : 'N U T, 0, 0, 0',
	X =  294.100  mm,	Y =   -361.050  mm,	Z =   -309.100  mm,
	W =  90.000 deg,	P =   0.000 deg,	R =   90.000 deg
};
P[2388]{
   GP1:
	UF : 0, UT : 6,		CONFIG : 'N U T, 0, 0, 0',
	X =  294.084  mm,	Y =   -361.159  mm,	Z =   -320.252  mm,
	W =  90.000 deg,	P =   0.000 deg,	R =   90.000 deg
};
P[2389]{
   GP1:
	UF : 0, UT : 6,		CONFIG : 'N U T, 0, 0, 0',
	X =  293.687  mm,	Y =   -361.131  mm,	Z =   -318.125  mm,
	W =  90.000 deg,	P =   0.000 deg,	R =   90.000 deg
};
P[2390]{
   GP1:
	UF : 0, UT : 6,		CONFIG : 'N U T, 0, 0, 0',
	X =  293.191  mm,	Y =   -361.206  mm,	Z =   -309.000  mm,
	W =  90.000 deg,	P =   0.000 deg,	R =   90.000 deg
};
P[2391]{
   GP1:
	UF : 0, UT : 6,		CONFIG : 'N U T, 0, 0, 0',
	X =  293.329  mm,	Y =   -361.655  mm,	Z =   -309.100  mm,
	W =  90.000 deg,	P =   0.000 deg,	R =   90.000 deg
};
P[2392]{
   GP1:
	UF : 0, UT : 6,		CONFIG : 'N U T, 0, 0, 0',
	X =  292.775  mm,	Y =   -361.749  mm,	Z =   -309.000  mm,
	W =  90.000 deg,	P =   0.000 deg,	R =   90.000 deg
};
P[2393]{
   GP1:
	UF : 0, UT : 6,		CONFIG : 'N U T, 0, 0, 0',
	X =  292.722  mm,	Y =   -362.104  mm,	Z =   -309.000  mm,
	W =  90.000 deg,	P =   0.000 deg,	R =   90.000 deg
};
P[2394]{
   GP1:
	UF : 0, UT : 6,		CONFIG : 'N U T, 0, 0, 0',
	X =  291.618  mm,	Y =   -362.596  mm,	Z =   -309.000  mm,
	W =  90.000 deg,	P =   0.000 deg,	R =   90.000 deg
};
P[2395]{
   GP1:
	UF : 0, UT : 6,		CONFIG : 'N U T, 0, 0, 0',
	X =  291.046  mm,	Y =   -363.231  mm,	Z =   -309.000  mm,
	W =  90.000 deg,	P =   0.000 deg,	R =   90.000 deg
};
P[2396]{
   GP1:
	UF : 0, UT : 6,		CONFIG : 'N U T, 0, 0, 0',
	X =  290.129  mm,	Y =   -363.633  mm,	Z =   -309.100  mm,
	W =  90.000 deg,	P =   0.000 deg,	R =   90.000 deg
};
P[2397]{
   GP1:
	UF : 0, UT : 6,		CONFIG : 'N U T, 0, 0, 0',
	X =  289.257  mm,	Y =   -363.485  mm,	Z =   -309.000  mm,
	W =  90.000 deg,	P =   0.000 deg,	R =   90.000 deg
};
P[2398]{
   GP1:
	UF : 0, UT : 6,		CONFIG : 'N U T, 0, 0, 0',
	X =  289.157  mm,	Y =   -364.058  mm,	Z =   -309.000  mm,
	W =  90.000 deg,	P =   0.000 deg,	R =   90.000 deg
};
P[2399]{
   GP1:
	UF : 0, UT : 6,		CONFIG : 'N U T, 0, 0, 0',
	X =  288.216  mm,	Y =   -364.285  mm,	Z =   -309.000  mm,
	W =  90.000 deg,	P =   0.000 deg,	R =   90.000 deg
};
P[2400]{
   GP1:
	UF : 0, UT : 6,		CONFIG : 'N U T, 0, 0, 0',
	X =  287.722  mm,	Y =   -364.682  mm,	Z =   -309.000  mm,
	W =  90.000 deg,	P =   0.000 deg,	R =   90.000 deg
};
P[2401]{
   GP1:
	UF : 0, UT : 6,		CONFIG : 'N U T, 0, 0, 0',
	X =  286.986  mm,	Y =   -364.616  mm,	Z =   -309.100  mm,
	W =  90.000 deg,	P =   0.000 deg,	R =   90.000 deg
};
P[2402]{
   GP1:
	UF : 0, UT : 6,		CONFIG : 'N U T, 0, 0, 0',
	X =  287.324  mm,	Y =   -365.232  mm,	Z =   -309.000  mm,
	W =  90.000 deg,	P =   0.000 deg,	R =   90.000 deg
};
P[2403]{
   GP1:
	UF : 0, UT : 6,		CONFIG : 'N U T, 0, 0, 0',
	X =  286.378  mm,	Y =   -365.388  mm,	Z =   -309.000  mm,
	W =  90.000 deg,	P =   0.000 deg,	R =   90.000 deg
};
P[2404]{
   GP1:
	UF : 0, UT : 6,		CONFIG : 'N U T, 0, 0, 0',
	X =  284.781  mm,	Y =   -366.233  mm,	Z =   -309.100  mm,
	W =  90.000 deg,	P =   0.000 deg,	R =   90.000 deg
};
P[2405]{
   GP1:
	UF : 0, UT : 6,		CONFIG : 'N U T, 0, 0, 0',
	X =  283.547  mm,	Y =   -367.168  mm,	Z =   -310.871  mm,
	W =  90.000 deg,	P =   0.000 deg,	R =   90.000 deg
};
P[2406]{
   GP1:
	UF : 0, UT : 6,		CONFIG : 'N U T, 0, 0, 0',
	X =  282.719  mm,	Y =   -367.409  mm,	Z =   -309.100  mm,
	W =  90.000 deg,	P =   0.000 deg,	R =   90.000 deg
};
P[2407]{
   GP1:
	UF : 0, UT : 6,		CONFIG : 'N U T, 0, 0, 0',
	X =  282.121  mm,	Y =   -368.198  mm,	Z =   -309.000  mm,
	W =  90.000 deg,	P =   0.000 deg,	R =   90.000 deg
};
P[2408]{
   GP1:
	UF : 0, UT : 6,		CONFIG : 'N U T, 0, 0, 0',
	X =  280.793  mm,	Y =   -368.737  mm,	Z =   -309.000  mm,
	W =  90.000 deg,	P =   0.000 deg,	R =   90.000 deg
};
P[2409]{
   GP1:
	UF : 0, UT : 6,		CONFIG : 'N U T, 0, 0, 0',
	X =  279.749  mm,	Y =   -368.956  mm,	Z =   -309.000  mm,
	W =  90.000 deg,	P =   0.000 deg,	R =   90.000 deg
};
P[2410]{
   GP1:
	UF : 0, UT : 6,		CONFIG : 'N U T, 0, 0, 0',
	X =  278.625  mm,	Y =   -369.841  mm,	Z =   -309.000  mm,
	W =  90.000 deg,	P =   0.000 deg,	R =   90.000 deg
};
P[2411]{
   GP1:
	UF : 0, UT : 6,		CONFIG : 'N U T, 0, 0, 0',
	X =  277.540  mm,	Y =   -370.579  mm,	Z =   -309.000  mm,
	W =  90.000 deg,	P =   0.000 deg,	R =   90.000 deg
};
P[2412]{
   GP1:
	UF : 0, UT : 6,		CONFIG : 'N U T, 0, 0, 0',
	X =  276.219  mm,	Y =   -371.646  mm,	Z =   -309.100  mm,
	W =  90.000 deg,	P =   0.000 deg,	R =   90.000 deg
};
P[2413]{
   GP1:
	UF : 0, UT : 6,		CONFIG : 'N U T, 0, 0, 0',
	X =  274.939  mm,	Y =   -371.874  mm,	Z =   -309.000  mm,
	W =  90.000 deg,	P =   0.000 deg,	R =   90.000 deg
};
P[2414]{
   GP1:
	UF : 0, UT : 6,		CONFIG : 'N U T, 0, 0, 0',
	X =  274.271  mm,	Y =   -372.465  mm,	Z =   -309.000  mm,
	W =  90.000 deg,	P =   0.000 deg,	R =   90.000 deg
};
P[2415]{
   GP1:
	UF : 0, UT : 6,		CONFIG : 'N U T, 0, 0, 0',
	X =  273.478  mm,	Y =   -372.840  mm,	Z =   -309.000  mm,
	W =  90.000 deg,	P =   0.000 deg,	R =   90.000 deg
};
P[2416]{
   GP1:
	UF : 0, UT : 6,		CONFIG : 'N U T, 0, 0, 0',
	X =  272.646  mm,	Y =   -373.451  mm,	Z =   -309.100  mm,
	W =  90.000 deg,	P =   0.000 deg,	R =   90.000 deg
};
P[2417]{
   GP1:
	UF : 0, UT : 6,		CONFIG : 'N U T, 0, 0, 0',
	X =  270.987  mm,	Y =   -374.237  mm,	Z =   -309.000  mm,
	W =  90.000 deg,	P =   0.000 deg,	R =   90.000 deg
};
P[2418]{
   GP1:
	UF : 0, UT : 6,		CONFIG : 'N U T, 0, 0, 0',
	X =  270.216  mm,	Y =   -374.649  mm,	Z =   -309.100  mm,
	W =  90.000 deg,	P =   0.000 deg,	R =   90.000 deg
};
P[2419]{
   GP1:
	UF : 0, UT : 6,		CONFIG : 'N U T, 0, 0, 0',
	X =  269.716  mm,	Y =   -375.451  mm,	Z =   -309.000  mm,
	W =  90.000 deg,	P =   0.000 deg,	R =   90.000 deg
};
P[2420]{
   GP1:
	UF : 0, UT : 6,		CONFIG : 'N U T, 0, 0, 0',
	X =  268.687  mm,	Y =   -375.709  mm,	Z =   -319.599  mm,
	W =  90.000 deg,	P =   0.000 deg,	R =   90.000 deg
};
P[2421]{
   GP1:
	UF : 0, UT : 6,		CONFIG : 'N U T, 0, 0, 0',
	X =  267.470  mm,	Y =   -376.394  mm,	Z =   -309.000  mm,
	W =  90.000 deg,	P =   0.000 deg,	R =   90.000 deg
};
P[2422]{
   GP1:
	UF : 0, UT : 6,		CONFIG : 'N U T, 0, 0, 0',
	X =  266.433  mm,	Y =   -376.946  mm,	Z =   -309.100  mm,
	W =  90.000 deg,	P =   0.000 deg,	R =   90.000 deg
};
P[2423]{
   GP1:
	UF : 0, UT : 6,		CONFIG : 'N U T, 0, 0, 0',
	X =  265.292  mm,	Y =   -377.299  mm,	Z =   -309.000  mm,
	W =  90.000 deg,	P =   0.000 deg,	R =   90.000 deg
};
P[2424]{
   GP1:
	UF : 0, UT : 6,		CONFIG : 'N U T, 0, 0, 0',
	X =  264.671  mm,	Y =   -378.232  mm,	Z =   -310.595  mm,
	W =  90.000 deg,	P =   0.000 deg,	R =   90.000 deg
};
P[2425]{
   GP1:
	UF : 0, UT : 6,		CONFIG : 'N U T, 0, 0, 0',
	X =  263.699  mm,	Y =   -378.385  mm,	Z =   -309.100  mm,
	W =  90.000 deg,	P =   0.000 deg,	R =   90.000 deg
};
P[2426]{
   GP1:
	UF : 0, UT : 6,		CONFIG : 'N U T, 0, 0, 0',
	X =  262.205  mm,	Y =   -379.792  mm,	Z =   -312.313  mm,
	W =  90.000 deg,	P =   0.000 deg,	R =   90.000 deg
};
P[2427]{
   GP1:
	UF : 0, UT : 6,		CONFIG : 'N U T, 0, 0, 0',
	X =  261.485  mm,	Y =   -379.851  mm,	Z =   -309.000  mm,
	W =  90.000 deg,	P =   0.000 deg,	R =   90.000 deg
};
P[2428]{
   GP1:
	UF : 0, UT : 6,		CONFIG : 'N U T, 0, 0, 0',
	X =  260.377  mm,	Y =   -380.168  mm,	Z =   -309.100  mm,
	W =  90.000 deg,	P =   0.000 deg,	R =   90.000 deg
};
P[2429]{
   GP1:
	UF : 0, UT : 6,		CONFIG : 'N U T, 0, 0, 0',
	X =  259.405  mm,	Y =   -381.156  mm,	Z =   -309.000  mm,
	W =  90.000 deg,	P =   0.000 deg,	R =   90.000 deg
};
P[2430]{
   GP1:
	UF : 0, UT : 6,		CONFIG : 'N U T, 0, 0, 0',
	X =  258.627  mm,	Y =   -381.472  mm,	Z =   -309.000  mm,
	W =  90.000 deg,	P =   0.000 deg,	R =   90.000 deg
};
P[2431]{
   GP1:
	UF : 0, UT : 6,		CONFIG : 'N U T, 0, 0, 0',
	X =  258.224  mm,	Y =   -382.285  mm,	Z =   -309.000  mm,
	W =  90.000 deg,	P =   0.000 deg,	R =   90.000 deg
};
P[2432]{
   GP1:
	UF : 0, UT : 6,		CONFIG : 'N U T, 0, 0, 0',
	X =  257.594  mm,	Y =   -381.993  mm,	Z =   -309.000  mm,
	W =  90.000 deg,	P =   0.000 deg,	R =   90.000 deg
};
P[2433]{
   GP1:
	UF : 0, UT : 6,		CONFIG : 'N U T, 0, 0, 0',
	X =  257.164  mm,	Y =   -382.696  mm,	Z =   -309.000  mm,
	W =  90.000 deg,	P =   0.000 deg,	R =   90.000 deg
};
P[2434]{
   GP1:
	UF : 0, UT : 6,		CONFIG : 'N U T, 0, 0, 0',
	X =  256.408  mm,	Y =   -382.955  mm,	Z =   -309.000  mm,
	W =  90.000 deg,	P =   0.000 deg,	R =   90.000 deg
};
P[2435]{
   GP1:
	UF : 0, UT : 6,		CONFIG : 'N U T, 0, 0, 0',
	X =  255.290  mm,	Y =   -383.568  mm,	Z =   -309.100  mm,
	W =  90.000 deg,	P =   0.000 deg,	R =   90.000 deg
};
P[2436]{
   GP1:
	UF : 0, UT : 6,		CONFIG : 'N U T, 0, 0, 0',
	X =  253.910  mm,	Y =   -384.605  mm,	Z =   -309.100  mm,
	W =  90.000 deg,	P =   0.000 deg,	R =   90.000 deg
};
P[2437]{
   GP1:
	UF : 0, UT : 6,		CONFIG : 'N U T, 0, 0, 0',
	X =  253.057  mm,	Y =   -385.129  mm,	Z =   -309.000  mm,
	W =  90.000 deg,	P =   0.000 deg,	R =   90.000 deg
};
P[2438]{
   GP1:
	UF : 0, UT : 6,		CONFIG : 'N U T, 0, 0, 0',
	X =  251.743  mm,	Y =   -385.283  mm,	Z =   -309.000  mm,
	W =  90.000 deg,	P =   0.000 deg,	R =   90.000 deg
};
P[2439]{
   GP1:
	UF : 0, UT : 6,		CONFIG : 'N U T, 0, 0, 0',
